(* If simulation of input enabled set it's value to FALSE *)
IF bResetForceValue THEN
	bResetForceValue := FALSE;
	piTestSensor.MR_ResetForceValue();
END_IF

bErrorTimedout := piTestSensor.ErrorTimedout;

bActive 		:= piTestSensor.Active;
CurrentTimeout	:= piTestSensor.CurrentTimeout;

IF bReset THEN
	bReset := FALSE;
	iState := 30;		
END_IF

CASE iState OF 
	0:
		IF bInit THEN
			bInit := FALSE;
			iState := 10;
			
		ELSIF bAbort THEN
			bAbort := FALSE;
			iState := 20;
			
		ELSIF bStartTracking THEN
			bStartTracking := FALSE;
			iState := 40;
			
		END_IF
	10:
		piTestSensor.MR_Init();
		IF piTestSensor.Active THEN
			iState := 0;
		END_IF
		
	20:
		piTestSensor.MR_Abort();
		IF NOT piTestSensor.Active THEN
			iState := 0;
		END_IF
		
	30:
		piTestSensor.MR_Reset();		
		IF NOT piTestSensor.ErrorTimedout THEN
			iState := 0;
		END_IF

	40:
		piTestSensor.MR_StartTracking();
		IF piTestSensor.In OR piTestSensor.ErrorTimedout THEN
			iState := 0;
		END_IF
	
END_CASE

piTestSensor();

END_PROGRAM

// ---- POUs/Universal Blocks/Digital Devices/Digital Output/PRG_FB_DigitalOutput_Test.TcPOU
PROGRAM PRG_FB_DigitalOutput_Test
VAR
	bFirstCycle		: BOOL := TRUE;
	bValue			: BOOL;					(* Output value to set on object *)
	poTestOutput	: FB_DigitalOutput();	(* Digital output object *)
END_VAR

IF bFirstCycle THEN
	bFirstCycle := FALSE;
	poTestOutput.MR_FirstCycle('My test digital output');
END_IF

poTestOutput.Out := bValue;
poTestOutput();

END_PROGRAM

// ---- POUs/Universal Blocks/Digital Devices/Lamp/PRG_FB_Lamp_Test.TcPOU
PROGRAM PRG_FB_Lamp_Test
VAR
	bFirstCycle 	: BOOL := TRUE;
	bTurnOn			: BOOL;				(* Command turn on *)
	bTurnOff		: BOOL;				(* Command turn off *)
	bStartFlashing	: BOOL;				(* Command start flashing *)
	tBlinkTime		: TIME := T#500MS;	(* Blink time *)
	fbLamp 			: FB_Lamp;			(* Lamp object *)
END_VAR

IF bFirstCycle THEN
	bFirstCycle := FALSE;
	fbLamp.MR_FirstCycle('My test lamp');
END_IF

IF bTurnOn THEN
	IF fbLamp.MR_LampOn() THEN
		bTurnOn := FALSE;
	END_IF
	
ELSIF bTurnOff THEN
	IF fbLamp.MR_LampOff() THEN
		bTurnOff := FALSE;
	END_IF
	
ELSIF bStartFlashing THEN
	IF fbLamp.MR_LampBlink(tBlinkTime) THEN
		bStartFlashing := FALSE;
	END_IF
	
END_IF

fbLamp();

END_PROGRAM

// ---- POUs/Universal Blocks/Fixtures/FB_Fixture222.TcPOU
FUNCTION_BLOCK FB_Fixture222 EXTENDS FB_UniversalFixture
VAR_INPUT
END_VAR
VAR_OUTPUT
END_VAR
VAR
	(*
		Add fixture sensors and actuators
	*)
END_VAR

SUPER^();

(*
	Add FB instances
*)

METHOD PROTECTED MS_Close
VAR_INPUT
END_VAR
eFixtureState := UNIVERSAL_FIXTURE_CLOSE_DONE;
END_METHOD

METHOD PROTECTED MS_Open
VAR_INPUT
END_VAR
eFixtureState := UNIVERSAL_FIXTURE_OPEN_DONE;
END_METHOD

METHOD PROTECTED MS_ReadyInitialized
VAR_INPUT
END_VAR
eFixtureState := UNIVERSAL_FIXTURE_IDLE;
END_METHOD

METHOD PROTECTED MS_Reset
VAR_INPUT
END_VAR
eFixtureState := UNIVERSAL_FIXTURE_RESET_DONE;
END_METHOD

PROPERTY SocketOpen : REFERENCE TO BOOL
GET
SocketOpen REF= bSocketOpen;
END_GET
END_PROPERTY

END_FUNCTION_BLOCK

// ---- POUs/Universal Blocks/Fixtures/PRG_FB_FixtureCommTest.TcPOU
PROGRAM PRG_FB_FixtureCommTest
VAR
	bFirstCycle			: BOOL := TRUE;
	
	(* Commands *)
	bInit				: BOOL;
	bMeasure 			: BOOL;
	bAbort				: BOOL;
	bReset				: BOOL;
	bOpen				: BOOL;
	bClose				: BOOL;
	
	(* Parameters *)
	iSampleID			: UINT;
	iState				: INT;
	
	(* Status *)
	bActive				: REFERENCE TO BOOL;
	bSocketOpen			: REFERENCE TO BOOL;
	iCurrentSampleID	: REFERENCE TO UDINT;
	bError				: REFERENCE TO BOOL;
	eFixtureState		: REFERENCE TO E_UniversalFixtureState;
	eResult				: REFERENCE TO E_UniversalFixtureSampleResult;
	
	(* FB's*)
	fbFixtureCommTest	: FB_Fixture;
END_VAR

IF bFirstCycle THEN
	bFirstCycle := FALSE;
	fbFixtureCommTest.MR_FirstCycle( 	sFixtureName 		:= 'PShEll Test Fixture',
										sHost 				:= '192.168.1.1',
										sAmsNetID 			:= '',
										iPort 				:= 12000,
										tTimeout 			:= DEFAULT_ADS_TIMEOUT,
										bUseLogger			:= TRUE,
										bClientConnection 	:= TRUE,
										sLoggerName 		:= 'PShEll Test Fixture',
										sFileDir 			:= 'C:\TwinCAT\Tests\',
										sFileName 			:= 'FixtureCommTest',
										bCreateFileAtStart 	:= TRUE,
										bAddHeader			:= TRUE,
										bAddTimeStamp 		:= TRUE);
	
	(* Update auxilary status variables *)									
	bActive 			REF= fbFixtureCommTest.Active;
	eResult				REF= fbFixtureCommTest.SampleResult;
	bError 				REF= fbFixtureCommTest.Error;
	eFixtureState		REF= fbFixtureCommTest.State;
	iCurrentSampleID	REF= fbFixtureCommTest.SampleID;
	bSocketOpen			REF= fbFixtureCommTest.SocketOpen;
END_IF

IF bReset THEN
	bReset := FALSE;
	iState := 50;
	
ELSIF bAbort THEN
	bAbort := FALSE;
	iState := 60;
	
END_IF

CASE iState OF
	0:
		IF bInit THEN
			bInit := FALSE;
			iState := 10;
			
		ELSIF bMeasure THEN
			bMeasure := FALSE;
			iState := 20;
			
		ELSIF bOpen THEN
			bOpen := FALSE;
			iState := 30;
		
		ELSIF bClose THEN
			bClose := FALSE;
			iState := 40;
			
		END_IF
	10:
		fbFixtureCommTest.MR_Init();
		
		IF fbFixtureCommTest.Active THEN
			iState := 0;
		END_IF
	20:
		fbFixtureCommTest.MR_Measure(iSampleID);
		
		IF NOT fbFixtureCommTest.Busy THEN
			iSampleID := 0;
			iState := 0;
		END_IF
		
	30:
		fbFixtureCommTest.MR_Open();
		
		IF fbFixtureCommTest.SocketOpen THEN
			iState := 0;
		END_IF
		
	40:
		fbFixtureCommTest.MR_Close();
		
		IF NOT fbFixtureCommTest.SocketOpen THEN
			iState := 0;
		END_IF
		
	50:
		fbFixtureCommTest.MR_Reset();
		
		IF NOT fbFixtureCommTest.Error THEN
			iState := 0;
		END_IF
	
	60:
		fbFixtureCommTest.MR_Abort();
		
		IF NOT fbFixtureCommTest.Active THEN
			iState := 0;
		END_IF
	
END_CASE

fbMachineTime(bEnable := TRUE);
fbFixtureCommTest();

END_PROGRAM

// ---- POUs/Universal Blocks/Fixture/FB_Fixture.TcPOU
(*
Copyrights	: Precision Systems Engineering
Author		: ADBO
Date		: 07/2022
Description	: This function block extends standard functionality of FB_FixtureCore with platform pusher and product holder.
*)
FUNCTION_BLOCK FB_Fixture EXTENDS FB_FixtureJig
VAR CONSTANT
	(* Fixture platform cylinder default setup *)
	sCOVER_PUSHER_NAME						: STRING	:= 'Cover Pusher';	(* Platform pusher name *)
	tCOVER_PUSHER_OPEN_TIMEOUT				: TIME 		:= T#5S;			(* Platform pusher opening timeout *)
	tCOVER_PUSHER_CLOSE_TIMEOUT				: TIME 		:= T#5S;			(* Platform pusher closing timeout *)
	tCOVER_PUSHER_MOVE_DELAY 				: TIME 		:= T#0MS;			(* Platform pusher delay after position change *)
	
	(* Fixture product holder default setup *)
	sCLAMP_NAME								: STRING 	:= 'Clamp Pusher';	(* Product holder name *)
	tCLAMP_OPEN_TIMEOUT						: TIME 		:= T#5S;			(* Product holder opening timeout *)
	tCLAMP_CLOSE_TIMEOUT					: TIME 		:= T#5S;			(* Product holder closing timeout *)
	tCLAMP_MOVE_DELAY 						: TIME 		:= T#300MS;//750MS	(* Product holder delay after position change *)
	
	(* Norm loading keywords *)
	sNORM_LOAD_COMMAND						: STRING := 'LDNORM:';			(* Load norm command send from PLC to UTU*)
	sNORM_GSAMPLE_MEASURE_COMMAND			: STRING := 'MeasGSample';		(* Measure Golden sample command send from PLC to UTU after loading new norm *)	
	sNORM_LOAD_SUCCESS 						: STRING := 'OK';				(* Response from UTU: norm loaded successfull *)
	sNORM_LOAD_FAIL							: STRING := 'Fail';				(* Response from UTU: norm load failed *)
	sNORM_GS_REQUEST						: STRING := 'GS:';				(* UTU requests golden sample *)
 	
	(* UTU STATUS *)
	sUTU_STATUS_OK							: STRING := 'OK';
	sUTU_STATUS_NOK							: STRING := 'NOK';
	sUTU_STATUS_bBusy						: STRING := 'bBusy';
	sUTU_STATUS_BCHECKSETUP					: STRING := 'bCheckSetup';
	
	(* Measurement keywords *)
	sMEASUREMENT_START_COMMAND				: STRING := 'bStart$R$N';		(* Start measurement command send from PLC to UTU*)
	
	sMEASUREMENT_BUSY						: STRING := 'bBusy';			(* Response from UTU: measurement started *)
	sMEASUREMENT_FINISHED					: STRING := (*'bReady'; //*)'bDone';			(* Response from UTU: measurement passed *)
	sMEASUREMENT_GOOD_PRODUCT				: STRING := 'bGood';			(* Response from UTU: good product *)
	sMEASUREMENT_REWORK						: STRING := 'bRework';			(* Perform remeasurement of same product *)
	sMEASUREMENT_REMEASURE					: STRING := 'bRemeasure';		(* Perform remeasurement of same product *)
	sMEASUREMENT_ERROR_THD					: STRING := 'bTHDReject';		(* Response from UTU: measurement failed with THD error*)
	sMEASUREMENT_ERROR_PHASE				: STRING := 'bPhaseReject';		(* Response from UTU: measurement failed with PHASE error*)
	sMEASUREMENT_ERROR_SSPL					: STRING := 'bSSPLReject';		(* Response from UTU: measurement failed with SSPL error*)
	sMEASUREMENT_ERROR_RUBBING				: STRING := 'bRubReject';		(* Response from UTU: measurement failed with RUBBING error*)
	sMEASUREMENT_ERROR_IMP					: STRING := 'bImpReject';		(* Response from UTU: measurement failed with INP error*)
	sMEASUREMENT_ERROR_HFA					: STRING := 'bHFAReject';		(* Response from UTU: measurement failed with HFA error*)
	sMEASUREMENT_ERROR_SPL					: STRING := 'bSPLReject';		(* Response from UTU: measurement failed with SPL error*)
	sMEASUREMENT_ERROR_CONNECTION			: STRING := 'bRejectConnect';	(* Response from UTU: measurement failed with connection problems *)
	sMEASUREMENT_ERROR_OTHER				: STRING := 'bReject';			(* Response from UTU: measurement failed *)
	sMEASUREMENT_FINISH_BATCH				: STRING := 'bFinishBatch';		(* Response from UTU: Batch END *)
	sMEASUREMENT_READY						: STRING := 'bReady';
END_VAR
VAR
	(* Auxilary command bits *)
	bCoverActive 							: BOOL;
	bCoverHome 								: BOOL;
	bClampHold 								: BOOL;
	bClampRelease 							: BOOL;
	bCoverActiveAndJigOpen					: BOOL;
	bCoverHomeAndJigClose					: BOOL;
	bLoadNorm								: BOOL;
//	bGSampleMeasure							: BOOL;
//	bGoldenSampelReadyToMeasure				: BOOL;		(* Robot gived Golden sample to Fixture *)
	
	(* Parameters *)
	sProductType							: STRING;
	sProductQuantity						: STRING;
	
	//new
	sConfig									: STRING;
	iAmount									: UINT;
	sPO										: STRING;
	sBatch									: STRING;
	sOPID									: STRING;
	
	(* Status flags *)
	bNormLoaded								: BOOL;
	bBatchEnd								: BOOL;
	bGSampleMeasureRequested				: BOOL;
	bReMeasure								: BOOL;
	bGSampleMeasurmentDone					: BOOL;
	eNormLoadResult							: E_FixtureLoadNormResult;
	eMeasurementResultExt					: E_FixtureMeasurementResultExt;
	
	(* State machines *)
	eFcqFixtureStateInit					: E_FixtureStateInit;
	eFcqFixtureStateAbort					: E_FixtureStateAbort;
	eFcqFixtrueStateReset					: E_FixtureStateReset;
	eFcqFixtureState						: E_FixtureState;
	eFcqFixtureStateLoadNorm				: E_FixtureStateLoadNorm;
	eFcqFixtureStateGSampleMeas				: E_FcqFixtureStateGSampleMeas;
	eFcqFixtureStateMeasurement 			: E_FixtureStateMeasurement;
	eFcqFixtureStateMeasurementDataExchange	: E_FixtureStateMeasurementDataExchange;
	
	eGoldenSampleResult 					: E_GoldenSampleState;
	
	iGsampleId : USINT;
	
	
	(* FB's *)
	fbCover									: FB_DoubleCoilCylinder;		(*  *)
	fbClamp									: FB_FixtureClamp;				(*  *)
	
END_VAR

IF bFirstCycle THEN
	fbCover.MR_FirstCycle(	sName 					:= CONCAT(STR1 :=THIS^.sName, STR2:= sCOVER_PUSHER_NAME),
							sHomeSensorModuleType	:= '?',
							sHomeSensorPortID		:= '?',
							sActiveSensorModuleType	:= '?',
							sActiveSensorPortID		:= '?',
							tGoHomeTimeout 			:= tCOVER_PUSHER_OPEN_TIMEOUT,
							tGoActiveTimeout 		:= tCOVER_PUSHER_CLOSE_TIMEOUT,
							tDelay					:= tCOVER_PUSHER_MOVE_DELAY);
									
	fbClamp.MR_FirstCycle(	sName 					:= CONCAT(STR1 := THIS^.sName, STR2:= sCLAMP_NAME),
							sHomeSensorModuleType	:= '?',
							sHomeSensorPortID		:= '?',
							sActiveSensorModuleType := '?',
							sActiveSensorPortID		:= '?',
							tGoHomeTimeout 			:= tCLAMP_OPEN_TIMEOUT,
							tGoActiveTimeout 		:= tCLAMP_CLOSE_TIMEOUT,
							tDelay					:= tCLAMP_MOVE_DELAY);							
END_IF

(* Run parent main implementation *)
SUPER^();

(* Update status flags*)
bError := bError OR fbClamp.Error OR fbCover.Error;
//IF bError THEN
//	bBusy := FALSE;
//END_IF

(* Run product holder cylinder instance *)
fbClamp();

(* Run fixture platform cylinder instance *)
fbCover();

PROPERTY BatchEnd : REFERENCE TO BOOL
GET
BatchEnd REF= bBatchEnd;
END_GET
END_PROPERTY

PROPERTY ClampHold : REFERENCE TO BOOL
GET
ClampHold REF= fbClamp.PositionActive;
//ClampHold := NOT fbClamp.PositionActive;
END_GET
END_PROPERTY

PROPERTY ClampSimulation : BOOL
GET
ClampSimulation := fbClamp.Simulation;
END_GET
SET
fbClamp.Simulation := ClampSimulation;
END_SET
END_PROPERTY

PROPERTY CoverPositionActive : REFERENCE TO BOOL
GET
CoverPositionActive REF= fbCover.PositionActive;
END_GET
END_PROPERTY

PROPERTY CoverPositionHome : REFERENCE TO BOOL
GET
CoverPositionHome REF= fbCover.PositionHome;
END_GET
END_PROPERTY

PROPERTY CoverSimulation : BOOL
GET
CoverSimulation := fbCover.Simulation;
END_GET
SET
fbCover.Simulation := CoverSimulation;
END_SET
END_PROPERTY

PROPERTY GoldenSampleMeasDone : REFERENCE TO BOOL
GET
GoldenSampleMeasDone REF= bGSampleMeasurmentDone;
END_GET
END_PROPERTY

PROPERTY GoldenSampleMeasRequested : REFERENCE TO BOOL
GET
GoldenSampleMeasRequested REF= bGSampleMeasureRequested;
END_GET
END_PROPERTY

PROPERTY GoldenSampleResult : REFERENCE TO E_GoldenSampleState
GET
GoldenSampleResult REF= eGoldenSampleResult;
END_GET
END_PROPERTY

PROPERTY GSampleId : REFERENCE TO USINT
GET
GSampleId REF= iGsampleId;
END_GET
END_PROPERTY

METHOD PROTECTED M_MeasurementClient : BOOL
VAR_INST
	tonMeasSimulation : TON;
END_VAR
CASE eFixtureStateMeasure OF
	UNIVERSAL_FIXTURE_MEASURE_SEND_DATA:
		sSendData := sMEASUREMENT_START_COMMAND;
		FUN_StringToTcpBufferData(sMessageAddr := ADR(sSendData), stSendDataAddr := ADR(stSendData));
		fbTcpClient.MR_AppendToSendBuffer(stData := stSendData);
		
		eFixtureStateMeasure := UNIVERSAL_FIXTURE_MEASURE_RECIVE_DATA;
		eFcqFixtureStateMeasurementDataExchange := FIXTURE_MEASURE_DATA_EXCHANGING_WAIT_FOR_BUSY;
		
	UNIVERSAL_FIXTURE_MEASURE_RECIVE_DATA:
		stReciveData := fbTcpClient.NextRecivedMessage;
		
		IF stReciveData.iLength > 0 THEN
			FUN_TcpBufferDataToString(sMessageAddr := ADR(sRecivedData), stReturnDataAddr := ADR(stReciveData));
		END_IF
		
			CASE eFcqFixtureStateMeasurementDataExchange OF
				FIXTURE_MEASURE_DATA_EXCHANGING_WAIT_FOR_BUSY:
					IF MEMCMP(ADR(sRecivedData),ADR(sMEASUREMENT_BUSY),INT_TO_UDINT(LEN(sMEASUREMENT_BUSY))) = 0 THEN
						fbTcpClient.MR_ClearReciveBuffer();
						eFcqFixtureStateMeasurementDataExchange := FIXTURE_MEASURE_DATA_EXCHANGING_WAIT_FOR_FISNISH;
					//	eFcqFixtureStateMeasurementDataExchange := FIXTURE_MEASURE_DATA_EXCHANGING_PROCCESS_RESULTS;
					END_IF
				
				FIXTURE_MEASURE_DATA_EXCHANGING_WAIT_FOR_FISNISH:
					IF (MEMCMP(ADR(sRecivedData),ADR(sMEASUREMENT_FINISHED),INT_TO_UDINT(LEN(sMEASUREMENT_FINISHED))) = 0) OR (FIND(sRecivedData,sMEASUREMENT_FINISHED) > 0) THEN
						IF bReMeasure THEN
							fbTcpClient.MR_ClearReciveBuffer();
							eFixtureStateMeasure := UNIVERSAL_FIXTURE_MEASURE_SEND_DATA;
							eFcqFixtureStateMeasurementDataExchange := FIXTURE_MEASURE_DATA_EXCHANGING_WAIT_FOR_BUSY;
						ELSE
							eFcqFixtureStateMeasurementDataExchange := FIXTURE_MEASURE_DATA_EXCHANGING_PROCCESS_RESULTS;
//							eFcqFixtureStateMeasurementDataExchange := FIXTURE_MEASURE_DATA_EXCHANGING_DONE;//
						END_IF	
					END_IF
				
				FIXTURE_MEASURE_DATA_EXCHANGING_PROCCESS_RESULTS:
					(* Good product *)
					IF (MEMCMP(ADR(sRecivedData),ADR(sMEASUREMENT_GOOD_PRODUCT),INT_TO_UDINT(LEN(sMEASUREMENT_GOOD_PRODUCT))) = 0) OR (FIND(sRecivedData,sMEASUREMENT_GOOD_PRODUCT) > 0) THEN
						IF bUseLogger THEN
							sLoggerMessage := CONCAT(sLoggerMessage,sMEASUREMENT_GOOD_PRODUCT);
							fbMeasurementLogger.MR_AddLogs(sLoggerMessage);
						END_IF
						fbTcpClient.MR_ClearReciveBuffer();
						eSampleResult := UNIVERSAL_FIXTURE_SAMPLE_ACCEPTED;
						eMeasurementResultExt := FIXTURE_MEASUREMENT_RESULT_GOOD;
						eFcqFixtureStateMeasurementDataExchange := FIXTURE_MEASURE_DATA_EXCHANGING_DONE;
//						eFcqFixtureStateMeasurementDataExchange := FIXTURE_MEASURE_DATA_EXCHANGING_WAIT_FOR_FISNISH; //

					(* Bad product - rework *)
					ELSIF (MEMCMP(ADR(sRecivedData),ADR(sMEASUREMENT_REWORK),INT_TO_UDINT(LEN(sMEASUREMENT_REWORK))) = 0) OR (FIND(sRecivedData,sMEASUREMENT_REWORK) > 0) THEN
						IF bUseLogger THEN
							sLoggerMessage := CONCAT(sLoggerMessage,sMEASUREMENT_REWORK);
							fbMeasurementLogger.MR_AddLogs(sLoggerMessage);
						END_IF
						fbTcpClient.MR_ClearReciveBuffer();
						eSampleResult := UNIVERSAL_FIXTURE_SAMPLE_REJECTED;
						eMeasurementResultExt := FIXTURE_MEASUREMENT_RESULT_REWORK;
						eFcqFixtureStateMeasurementDataExchange := FIXTURE_MEASURE_DATA_EXCHANGING_DONE;
//						eFcqFixtureStateMeasurementDataExchange := FIXTURE_MEASURE_DATA_EXCHANGING_WAIT_FOR_FISNISH; //
						
						
					(* Bad product - remeaseure *)
					ELSIF (MEMCMP(ADR(sRecivedData),ADR(sMEASUREMENT_REMEASURE),INT_TO_UDINT(LEN(sMEASUREMENT_REMEASURE))) = 0) OR (FIND(sRecivedData,sMEASUREMENT_REMEASURE) > 0) THEN
						fbTcpClient.MR_ClearSendBuffer();
						fbTcpClient.MR_ClearReciveBuffer();
//						bReMeasure := TRUE;
//						eFcqFixtureStateMeasurementDataExchange :=FIXTURE_MEASURE_DATA_EXCHANGING_WAIT_FOR_FISNISH;
						eFixtureStateMeasure := UNIVERSAL_FIXTURE_MEASURE_SEND_DATA;
						eFcqFixtureStateMeasurementDataExchange := FIXTURE_MEASURE_DATA_EXCHANGING_WAIT_FOR_BUSY;
						
					(* Bad product - connection *)	
					ELSIF (MEMCMP(ADR(sRecivedData),ADR(sMEASUREMENT_ERROR_CONNECTION),INT_TO_UDINT(LEN(sMEASUREMENT_ERROR_CONNECTION))) = 0) OR  (FIND(sRecivedData,sMEASUREMENT_ERROR_CONNECTION) > 0)  THEN
						IF bUseLogger THEN
							sLoggerMessage := CONCAT(sLoggerMessage,sMEASUREMENT_ERROR_CONNECTION);
							fbMeasurementLogger.MR_AddLogs(sLoggerMessage);
						END_IF
						fbTcpClient.MR_ClearReciveBuffer();
						eSampleResult := UNIVERSAL_FIXTURE_SAMPLE_REJECTED;
						eMeasurementResultExt := FIXTURE_MEASUREMENT_RESULT_CONNECT;
						eFcqFixtureStateMeasurementDataExchange := FIXTURE_MEASURE_DATA_EXCHANGING_DONE;
//						eFcqFixtureStateMeasurementDataExchange := FIXTURE_MEASURE_DATA_EXCHANGING_WAIT_FOR_FISNISH; //
					
					(* Bad product - THD *)
					ELSIF (MEMCMP(ADR(sRecivedData),ADR(sMEASUREMENT_ERROR_THD),INT_TO_UDINT(LEN(sMEASUREMENT_ERROR_THD))) = 0) OR (FIND(sRecivedData,sMEASUREMENT_ERROR_THD) > 0)  THEN
						IF bUseLogger THEN
							sLoggerMessage := CONCAT(sLoggerMessage,sMEASUREMENT_ERROR_THD);
							fbMeasurementLogger.MR_AddLogs(sLoggerMessage);
						END_IF
						fbTcpClient.MR_ClearReciveBuffer();
						eSampleResult := UNIVERSAL_FIXTURE_SAMPLE_REJECTED;
						eMeasurementResultExt := (*FIXTURE_MEASUREMENT_RESULT_REWORK;*)FIXTURE_MEASUREMENT_RESULT_THD;
						eFcqFixtureStateMeasurementDataExchange := FIXTURE_MEASURE_DATA_EXCHANGING_DONE;
//						eFcqFixtureStateMeasurementDataExchange := FIXTURE_MEASURE_DATA_EXCHANGING_WAIT_FOR_FISNISH; //
					
					(* Bad product - PHASE *)
					ELSIF (MEMCMP(ADR(sRecivedData),ADR(sMEASUREMENT_ERROR_PHASE),INT_TO_UDINT(LEN(sMEASUREMENT_ERROR_PHASE))) = 0) OR (FIND(sRecivedData,sMEASUREMENT_ERROR_PHASE) > 0) THEN
						IF bUseLogger THEN
							sLoggerMessage := CONCAT(sLoggerMessage,sMEASUREMENT_ERROR_PHASE);
							fbMeasurementLogger.MR_AddLogs(sLoggerMessage);
						END_IF
						fbTcpClient.MR_ClearReciveBuffer();
						eSampleResult := UNIVERSAL_FIXTURE_SAMPLE_REJECTED;
						eMeasurementResultExt := FIXTURE_MEASUREMENT_RESULT_PHASE;
						eFcqFixtureStateMeasurementDataExchange := FIXTURE_MEASURE_DATA_EXCHANGING_DONE;
//						eFcqFixtureStateMeasurementDataExchange := FIXTURE_MEASURE_DATA_EXCHANGING_WAIT_FOR_FISNISH; //
					
					(* Bad product - SSPL *)
					ELSIF (MEMCMP(ADR(sRecivedData),ADR(sMEASUREMENT_ERROR_SSPL),INT_TO_UDINT(LEN(sMEASUREMENT_ERROR_SSPL))) = 0) OR (FIND(sRecivedData,sMEASUREMENT_ERROR_SSPL) > 0) THEN
						IF bUseLogger THEN
							sLoggerMessage := CONCAT(sLoggerMessage,sMEASUREMENT_ERROR_SSPL);
							fbMeasurementLogger.MR_AddLogs(sLoggerMessage);
						END_IF
						fbTcpClient.MR_ClearReciveBuffer();
						eSampleResult := UNIVERSAL_FIXTURE_SAMPLE_REJECTED;
						eMeasurementResultExt := FIXTURE_MEASUREMENT_RESULT_SSPL;
						eFcqFixtureStateMeasurementDataExchange := FIXTURE_MEASURE_DATA_EXCHANGING_DONE;
//						eFcqFixtureStateMeasurementDataExchange := FIXTURE_MEASURE_DATA_EXCHANGING_WAIT_FOR_FISNISH; //
					
					(* Bad product - Rubbing *)
					ELSIF (MEMCMP(ADR(sRecivedData),ADR(sMEASUREMENT_ERROR_RUBBING),INT_TO_UDINT(LEN(sMEASUREMENT_ERROR_RUBBING))) = 0) OR (FIND(sRecivedData,sMEASUREMENT_ERROR_RUBBING) > 0) THEN
						IF bUseLogger THEN
							sLoggerMessage := CONCAT(sLoggerMessage,sMEASUREMENT_ERROR_RUBBING);
							fbMeasurementLogger.MR_AddLogs(sLoggerMessage);
						END_IF
						fbTcpClient.MR_ClearReciveBuffer();
						eSampleResult := UNIVERSAL_FIXTURE_SAMPLE_REJECTED;
						eMeasurementResultExt := FIXTURE_MEASUREMENT_RESULT_RUBBING;
						eFcqFixtureStateMeasurementDataExchange := FIXTURE_MEASURE_DATA_EXCHANGING_DONE;
//						eFcqFixtureStateMeasurementDataExchange := FIXTURE_MEASURE_DATA_EXCHANGING_WAIT_FOR_FISNISH; //
					
					(* Bad product - IMP *)
					ELSIF (MEMCMP(ADR(sRecivedData),ADR(sMEASUREMENT_ERROR_IMP),INT_TO_UDINT(LEN(sMEASUREMENT_ERROR_IMP))) = 0) OR (FIND(sRecivedData,sMEASUREMENT_ERROR_IMP) > 0) THEN
						IF bUseLogger THEN
							sLoggerMessage := CONCAT(sLoggerMessage,sMEASUREMENT_ERROR_IMP);
							fbMeasurementLogger.MR_AddLogs(sLoggerMessage);
						END_IF
						fbTcpClient.MR_ClearReciveBuffer();
						eSampleResult := UNIVERSAL_FIXTURE_SAMPLE_REJECTED;
						eMeasurementResultExt := FIXTURE_MEASUREMENT_RESULT_IMP;
						eFcqFixtureStateMeasurementDataExchange := FIXTURE_MEASURE_DATA_EXCHANGING_DONE;
//						eFcqFixtureStateMeasurementDataExchange := FIXTURE_MEASURE_DATA_EXCHANGING_WAIT_FOR_FISNISH; //
					
					(* Bad product - HFA *)
					ELSIF (MEMCMP(ADR(sRecivedData),ADR(sMEASUREMENT_ERROR_HFA),INT_TO_UDINT(LEN(sMEASUREMENT_ERROR_HFA))) = 0) OR (FIND(sRecivedData,sMEASUREMENT_ERROR_HFA) > 0) THEN
						IF bUseLogger THEN
							sLoggerMessage := CONCAT(sLoggerMessage,sMEASUREMENT_ERROR_HFA);
							fbMeasurementLogger.MR_AddLogs(sLoggerMessage);
						END_IF
						fbTcpClient.MR_ClearReciveBuffer();
						eSampleResult := UNIVERSAL_FIXTURE_SAMPLE_REJECTED;
						eMeasurementResultExt := FIXTURE_MEASUREMENT_RESULT_HFA;
						eFcqFixtureStateMeasurementDataExchange := FIXTURE_MEASURE_DATA_EXCHANGING_DONE;
//						eFcqFixtureStateMeasurementDataExchange := FIXTURE_MEASURE_DATA_EXCHANGING_WAIT_FOR_FISNISH; //
						
					(* Bad product - SPL *)
					ELSIF (MEMCMP(ADR(sRecivedData),ADR(sMEASUREMENT_ERROR_OTHER),INT_TO_UDINT(LEN(sMEASUREMENT_ERROR_OTHER))) = 0) OR (FIND(sRecivedData,sMEASUREMENT_ERROR_OTHER) > 0) THEN
						IF bUseLogger THEN
							sLoggerMessage := CONCAT(sLoggerMessage,sMEASUREMENT_ERROR_SPL);
							fbMeasurementLogger.MR_AddLogs(sLoggerMessage);
						END_IF
						fbTcpClient.MR_ClearReciveBuffer();
						eSampleResult := UNIVERSAL_FIXTURE_SAMPLE_REJECTED;
						eMeasurementResultExt := FIXTURE_MEASUREMENT_RESULT_SPL;
						eFcqFixtureStateMeasurementDataExchange := FIXTURE_MEASURE_DATA_EXCHANGING_DONE;
//						eFcqFixtureStateMeasurementDataExchange := FIXTURE_MEASURE_DATA_EXCHANGING_WAIT_FOR_FISNISH; //
					
					ELSIF (MEMCMP(ADR(sRecivedData),ADR(sMEASUREMENT_ERROR_OTHER),INT_TO_UDINT(LEN(sMEASUREMENT_ERROR_OTHER))) = 0) OR (FIND(sRecivedData,sMEASUREMENT_ERROR_OTHER) > 0)  THEN
						IF bUseLogger THEN
							sLoggerMessage := CONCAT(sLoggerMessage,sMEASUREMENT_ERROR_OTHER);
							fbMeasurementLogger.MR_AddLogs(sLoggerMessage);
						END_IF
						fbTcpClient.MR_ClearReciveBuffer();
						eSampleResult := UNIVERSAL_FIXTURE_SAMPLE_REJECTED;
						eMeasurementResultExt := FIXTURE_MEASUREMENT_RESULT_REJECT_OTHER;
						eFcqFixtureStateMeasurementDataExchange := FIXTURE_MEASURE_DATA_EXCHANGING_DONE;
					
					ELSIF (MEMCMP(ADR(sRecivedData),ADR(sMEASUREMENT_READY),INT_TO_UDINT(LEN(sMEASUREMENT_READY))) = 0) OR (FIND(sRecivedData,sMEASUREMENT_READY) > 0)  THEN 
						eFcqFixtureStateMeasurementDataExchange := FIXTURE_MEASURE_DATA_EXCHANGING_DONE;	
					END_IF
					
				FIXTURE_MEASURE_DATA_EXCHANGING_DONE:
					IF (MEMCMP(ADR(sRecivedData),ADR(sMEASUREMENT_READY),INT_TO_UDINT(LEN(sMEASUREMENT_READY))) = 0) OR (FIND(sRecivedData,sMEASUREMENT_READY) > 0) THEN
						eFixtureStateMeasure := UNIVERSAL_FIXTURE_MEASURE_DONE;
					END_IF
			END_CASE		
	//	END_IF
	
	UNIVERSAL_FIXTURE_MEASURE_DONE:
		IF 	(MEMCMP(ADR(sRecivedData),ADR(sMEASUREMENT_FINISH_BATCH),INT_TO_UDINT(LEN(sMEASUREMENT_FINISH_BATCH))) = 0) OR (FIND(sRecivedData,sMEASUREMENT_FINISH_BATCH) > 0) THEN
			bBatchEnd := TRUE;
		END_IF
		fbTcpClient.MR_ClearAllBuffers();
		eFixtureState := UNIVERSAL_FIXTURE_METHOD_DONE;
		
END_CASE
(*
tonMeasSimulation(IN := TRUE, PT := T#2500MS);
IF tonMeasSimulation.Q THEN
	tonMeasSimulation(IN := FALSE);
	eSampleResult := UNIVERSAL_FIXTURE_SAMPLE_ACCEPTED;
	eMeasurementResultExt := FIXTURE_MEASUREMENT_RESULT_GOOD;
	eFixtureState := UNIVERSAL_FIXTURE_METHOD_DONE;
END_IF
*)
END_METHOD

PROPERTY MeasurementResultExt : REFERENCE TO E_FixtureMeasurementResultExt
GET
MeasurementResultExt REF= eMeasurementResultExt;
END_GET
END_PROPERTY

METHOD MR_ClampHold : BOOL
VAR_INPUT
END_VAR
IF eFixtureState = UNIVERSAL_FIXTURE_IDLE AND NOT fbClamp.PositionActive THEN
	bBusy := TRUE;
	bClampHold := TRUE;
	MR_ClampHold := FALSE;
	eFixtureState := UNIVERSAL_FIXTURE_EXTENSION;
	eFcqFixtureState := FIXTURE_EXTENSION_CLAMP_HOLD;
	fbMachineLogger.MR_AddLogs(CONCAT(sName,' : product hold'));
	
ELSIF eFcqFixtureState = FIXTURE_EXTENSION_CLAMP_HOLD_DONE THEN
	bClampHold := FALSE;
	MR_ClampHold := TRUE;
	fbMachineLogger.MR_AddLogs(CONCAT(sName,' : product hold done'));
	
END_IF
END_METHOD

METHOD MR_ClampRelease : BOOL
VAR_INPUT
END_VAR
IF eFixtureState = UNIVERSAL_FIXTURE_IDLE AND fbClamp.PositionActive THEN
	bBusy := TRUE;
	bClampRelease := TRUE;
	MR_ClampRelease := FALSE;
	eFixtureState := UNIVERSAL_FIXTURE_EXTENSION;
	eFcqFixtureState := FIXTURE_EXTENSION_CLAMP_RELEASE;
	fbMachineLogger.MR_AddLogs(CONCAT(sName,' : product release'));
	
ELSIF eFcqFixtureState = FIXTURE_EXTENSION_CLAMP_RELEASE_DONE THEN
	bClampRelease := FALSE;
	MR_ClampRelease := TRUE;
	fbMachineLogger.MR_AddLogs(CONCAT(sName,' : product release done'));
	
END_IF
END_METHOD

METHOD MR_CoverActive : BOOL
VAR_INPUT
END_VAR
IF eFixtureState = UNIVERSAL_FIXTURE_IDLE AND NOT fbCover.PositionActive THEN
	bBusy := TRUE;
	bCoverActive := TRUE;
	MR_CoverActive := FALSE;
	eFixtureState := UNIVERSAL_FIXTURE_EXTENSION;
	eFcqFixtureState := FIXTURE_EXTENSION_COVER_ACTIVE;
	fbMachineLogger.MR_AddLogs(CONCAT(sName,' : platform go active'));
	
ELSIF eFcqFixtureState = FIXTURE_EXTENSION_COVER_ACTIVE_DONE THEN
	bCoverActive := FALSE;
	MR_CoverActive := TRUE;
	fbMachineLogger.MR_AddLogs(CONCAT(sName,' : platform go active done'));
	
END_IF
END_METHOD

METHOD MR_CoverActiveAndJigOpen : BOOL
VAR_INPUT
END_VAR
//IF eFixtureState = UNIVERSAL_FIXTURE_IDLE AND (NOT fbCover.PositionActive AND NOT THIS^.SocketOpen) THEN
IF eFixtureState = UNIVERSAL_FIXTURE_IDLE AND (NOT fbCover.PositionActive OR NOT THIS^.SocketOpen) THEN
	bBusy := TRUE;
	bCoverActiveAndJigOpen := TRUE;
	MR_CoverActiveAndJigOpen := FALSE;
	eFixtureState := UNIVERSAL_FIXTURE_EXTENSION;
	eFcqFixtureState := FIXTURE_EXTENSION_COVER_ACTIVE_AND_JIG_OPEN;
	fbMachineLogger.MR_AddLogs(CONCAT(sName,' : platform go active and open'));
	
ELSIF eFcqFixtureState = FIXTURE_EXTENSION_COVER_ACTIVE_AND_JIG_OPEN_DONE THEN
	bCoverActiveAndJigOpen := FALSE;
	MR_CoverActiveAndJigOpen := TRUE;
	fbMachineLogger.MR_AddLogs(CONCAT(sName,' : platform go active and open done'));
	
END_IF
END_METHOD

METHOD MR_CoverHome : BOOL
VAR_INPUT
END_VAR
IF eFixtureState = UNIVERSAL_FIXTURE_IDLE AND NOT fbCover.PositionHome THEN
	bBusy := TRUE;
	bCoverHome := TRUE;
	MR_CoverHome := FALSE;
	eFixtureState := UNIVERSAL_FIXTURE_EXTENSION;
	eFcqFixtureState := FIXTURE_EXTENSION_COVER_HOME;
	fbMachineLogger.MR_AddLogs(CONCAT(sName,' : platform go home'));
	
ELSIF eFcqFixtureState = FIXTURE_EXTENSION_COVER_HOME_DONE THEN
	bCoverHome := FALSE;
	MR_CoverHome := TRUE;
	fbMachineLogger.MR_AddLogs(CONCAT(sName,' : platform go home done'));
	
END_IF
END_METHOD

METHOD MR_CoverHomeAndJigClose : BOOL
VAR_INPUT
END_VAR
//IF eFixtureState = UNIVERSAL_FIXTURE_IDLE AND NOT fbCover.PositionHome AND THIS^.SocketOpen THEN
IF eFixtureState = UNIVERSAL_FIXTURE_IDLE AND (NOT fbCover.PositionHome OR THIS^.SocketOpen) THEN
	bBusy := TRUE;
	bCoverHomeAndJigClose := TRUE;
	MR_CoverHomeAndJigClose := FALSE;
	eFixtureState := UNIVERSAL_FIXTURE_EXTENSION;
	eFcqFixtureState := FIXTURE_EXTENSION_COVER_HOME_AND_JIG_CLOSE;
	fbMachineLogger.MR_AddLogs(CONCAT(sName,' : platform go home and close'));
	
ELSIF eFcqFixtureState = FIXTURE_EXTENSION_COVER_HOME_AND_JIG_CLOSE_DONE THEN
	bCoverHomeAndJigClose := FALSE;
	MR_CoverHomeAndJigClose := TRUE;
	fbMachineLogger.MR_AddLogs(CONCAT(sName,' : platform go home and close done'));
	
END_IF
END_METHOD

METHOD MR_GSampleMeas : BOOL
VAR_INPUT
END_VAR
//IF eNormLoadResult = FIXTURE_NORM_LOAD_GOLDEN_SAMPLE_NEEDED AND eFcqFixtureStateLoadNorm = FIXTURE_LOADING_NORM_GOLDEN_SAMPLE_WAIT_FOR_END THEN
IF eNormLoadResult = FIXTURE_NORM_LOAD_GOLDEN_SAMPLE_NEEDED AND eFixtureState = UNIVERSAL_FIXTURE_IDLE THEN
	bBusy := TRUE;
	bGSampleMeasurmentDone := FALSE;	
	MR_GSampleMeas := FALSE;
//	bGSampleMeasure := TRUE;
	eGoldenSampleResult := GS_STATUS_UNKNOWN;
	eFixtureState := UNIVERSAL_FIXTURE_EXTENSION;
	eFcqFixtureState := FIXTURE_EXTENSION_GOLDEN_SAMPLE_MEASURE;
	eFcqFixtureStateGSampleMeas := FIXTURE_GOLDEN_SAMPLE_SEND_MEASURE_COMMAND;
	fbMachineLogger.MR_AddLogs(CONCAT(sName,' : Golden Sample measurment requested'));
	
	
ELSIF eFcqFixtureState = FIXTURE_EXTENSION_GOLDEN_SAMPLE_MEASURE_DONE THEN
	bBusy := FALSE;
	MR_GSampleMeas := TRUE;
	eFixtureState := UNIVERSAL_FIXTURE_EXTENSION;
	eFcqFixtureState := FIXTURE_EXTENSION_LOAD_NORM;
	//eFcqFixtureStateLoadNorm := FIXTURE_LOADING_NORM_WAIT_FOR_RESPONSE;
	//fbMachineLogger.MR_AddLogs(CONCAT(sName,' : Golden Sample  '));
	fbMachineLogger.MR_AddLogs(CONCAT(sName,CONCAT(' : Golden Sample ID: ',CONCAT(UDINT_TO_STRING(iGsampleId),' measurment done'))));
	bGSampleMeasurmentDone := TRUE;
END_IF
END_METHOD

METHOD MR_LoadNorm : BOOL
VAR_INPUT
	sConfig				: STRING;
	iAmount				: UINT;
	sPO					: STRING;
	sBatch				: STRING;
	sOPID				: STRING;
//	sProductType 		: STRING;	(* Name of product possesed from MES*)
//	sProductQuantity	: STRING;	(* Product quantity *)
END_VAR
IF eFixtureState = UNIVERSAL_FIXTURE_IDLE THEN
	THIS^.sConfig := sConfig;
	THIS^.iAmount := iAmount;
	THIS^.sPO := sPO;
	THIS^.sBatch := sBatch;
	THIS^.sOPID := sOPID;
	
(*	OLD
	THIS^.sProductType := sProductType;
	THIS^.sProductQuantity := sProductQuantity;
*)	
	bNormLoaded := FALSE;
	eNormLoadResult := FIXTURE_NORM_LOAD_UNKNOWN;
//	bLoadNorm := TRUE;
	MR_LoadNorm := FALSE;
	eFixtureState := UNIVERSAL_FIXTURE_EXTENSION;
	eFcqFixtureState := FIXTURE_EXTENSION_LOAD_NORM;
	eFcqFixtureStateLoadNorm := FIXTURE_LOADING_NORM_SEND_NORM_DATA;
	fbMachineLogger.MR_AddLogs(CONCAT(sName,' : load norm requested'));
	
ELSIF eFcqFixtureState = FIXTURE_EXTENSION_LOAD_NORM_DONE THEN
	bNormLoaded := (*NOT bGSampleMeasureRequested;//*)TRUE;
	MR_LoadNorm := TRUE;
	fbMachineLogger.MR_AddLogs(CONCAT(sName,' : norm loaded '));
	
END_IF
END_METHOD

METHOD MR_Reset : BOOL
VAR_INPUT
END_VAR
IF eFixtureState = UNIVERSAL_FIXTURE_METHOD_DONE THEN
	eFcqFixtrueStateReset:=FIXTURE_RESET_CLAMP;
END_IF
SUPER^.MR_Reset();
END_METHOD

METHOD PROTECTED MS_Aborting
VAR_INPUT
END_VAR
CASE eFcqFixtureStateAbort OF
	FIXTURE_ABORT_CLAMP:
		fbClamp.MR_Abort();
		IF NOT fbClamp.Active THEN
			eFcqFixtureStateAbort := FIXTURE_ABORT_COVER;
		END_IF
		
	FIXTURE_ABORT_COVER:
		fbCover.MR_Abort();
		IF NOT fbCover.Active THEN
			eJigStateAbort := FIXTURE_JIG_ABORT_JIG_PUSHER;
			eFcqFixtureStateAbort := FIXTURE_ABORT_DONE;
		END_IF
		
	FIXTURE_ABORT_DONE:
		SUPER^.MS_Aborting();
		
END_CASE
END_METHOD

METHOD MS_ClampHold
VAR_INPUT
END_VAR
fbClamp.MR_GoActive();
IF fbClamp.PositionActive AND NOT fbClamp.Busy THEN
	eFcqFixtureState := FIXTURE_EXTENSION_CLAMP_HOLD_DONE;
END_IF
END_METHOD

METHOD MS_ClampHoldDone
VAR_INPUT
END_VAR
IF NOT bClampHold THEN
	bBusy := FALSE;
	eFixtureState := UNIVERSAL_FIXTURE_IDLE;
	eFcqFixtureState := FIXTURE_EXTENSION_IDLE;
END_IF
END_METHOD

METHOD MS_ClampRelease
VAR_INPUT
END_VAR
fbClamp.MR_GoHome();
IF NOT fbClamp.PositionActive AND NOT fbClamp.Busy THEN
	eFcqFixtureState := FIXTURE_EXTENSION_CLAMP_RELEASE_DONE;
END_IF
END_METHOD

METHOD MS_ClampReleaseDone
VAR_INPUT
END_VAR
IF NOT bClampRelease THEN
	bBusy := FALSE;
	eFixtureState := UNIVERSAL_FIXTURE_IDLE;
	eFcqFixtureState := FIXTURE_EXTENSION_IDLE;
END_IF
END_METHOD

METHOD MS_CoverActive
VAR_INPUT
END_VAR
fbCover.MR_GoActive();
IF fbCover.PositionActive AND NOT fbCover.Busy THEN
	eFcqFixtureState := FIXTURE_EXTENSION_COVER_ACTIVE_DONE;
END_IF
END_METHOD

METHOD MS_CoverActiveAndJigOpen : BOOL
VAR_INPUT
END_VAR
fbCover.MR_GoActive();
fbJig.MR_GoActive();
IF fbCover.PositionActive AND NOT fbCover.Busy AND
	fbJig.PositionActive AND NOT fbJig.Busy THEN
	eFcqFixtureState := FIXTURE_EXTENSION_COVER_ACTIVE_AND_JIG_OPEN_DONE;
END_IF
END_METHOD

METHOD MS_CoverActiveAndJigOpenDone : BOOL
VAR_INPUT
END_VAR
IF NOT bCoverActiveAndJigOpen THEN
	bBusy := FALSE;
	eFixtureState := UNIVERSAL_FIXTURE_IDLE;
	eFcqFixtureState := FIXTURE_EXTENSION_IDLE;
END_IF
END_METHOD

METHOD MS_CoverActiveDone
VAR_INPUT
END_VAR
IF NOT bCoverActive THEN
	bBusy := FALSE;
	eFixtureState := UNIVERSAL_FIXTURE_IDLE;
	eFcqFixtureState := FIXTURE_EXTENSION_IDLE;
END_IF
END_METHOD

METHOD MS_CoverHome
VAR_INPUT
END_VAR
fbCover.MR_GoHome();
IF fbCover.PositionHome AND NOT fbCover.Busy THEN
	eFcqFixtureState := FIXTURE_EXTENSION_COVER_HOME_DONE;
END_IF
END_METHOD

METHOD MS_CoverHomeAndJigClose : BOOL
VAR_INPUT
END_VAR
fbCover.MR_GoHome();
fbJig.MR_GoHome();
IF fbCover.PositionHome AND NOT fbCover.Busy AND
	fbJig.PositionHome AND NOT fbJig.Busy THEN
	eFcqFixtureState := FIXTURE_EXTENSION_COVER_HOME_AND_JIG_CLOSE_DONE;
END_IF
END_METHOD

METHOD MS_CoverHomeAndJigCloseDone : BOOL
VAR_INPUT
END_VAR
IF NOT bCoverHomeAndJigClose THEN
	bBusy := FALSE;
	eFixtureState := UNIVERSAL_FIXTURE_IDLE;
	eFcqFixtureState := FIXTURE_EXTENSION_IDLE;
END_IF
END_METHOD

METHOD MS_CoverHomeDone
VAR_INPUT
END_VAR
IF NOT bCoverHome THEN
	bBusy := FALSE;
	eFixtureState := UNIVERSAL_FIXTURE_IDLE;
	eFcqFixtureState := FIXTURE_EXTENSION_IDLE;
END_IF
END_METHOD

METHOD PROTECTED MS_Extension
VAR_INPUT
END_VAR
CASE eFcqFixtureState OF
	E_FixtureState.FIXTURE_EXTENSION_IDLE:
		bBusy := FALSE;
		
	E_FixtureState.FIXTURE_EXTENSION_COVER_ACTIVE:
		MS_CoverActive();
		
	E_FixtureState.FIXTURE_EXTENSION_COVER_ACTIVE_DONE:
		MS_CoverActiveDone();
		
	E_FixtureState.FIXTURE_EXTENSION_COVER_HOME:
		MS_CoverHome();
		
	E_FixtureState.FIXTURE_EXTENSION_COVER_HOME_DONE:
		MS_CoverHomeDone();	
	
	E_FixtureState.FIXTURE_EXTENSION_CLAMP_HOLD:
		MS_ClampHold();
		
	E_FixtureState.FIXTURE_EXTENSION_CLAMP_HOLD_DONE:
		MS_ClampHoldDone();
		
	E_FixtureState.FIXTURE_EXTENSION_CLAMP_RELEASE:
		MS_ClampRelease();
		
	E_FixtureState.FIXTURE_EXTENSION_CLAMP_RELEASE_DONE:
		MS_ClampReleaseDone();
	
	FIXTURE_EXTENSION_COVER_ACTIVE_AND_JIG_OPEN:
		MS_CoverActiveAndJigOpen();
		
	FIXTURE_EXTENSION_COVER_ACTIVE_AND_JIG_OPEN_DONE:
		MS_CoverActiveAndJigOpenDone();
		
	FIXTURE_EXTENSION_COVER_HOME_AND_JIG_CLOSE:
		MS_CoverHomeAndJigClose();
		
	FIXTURE_EXTENSION_COVER_HOME_AND_JIG_CLOSE_DONE:
		MS_CoverHomeAndJigCloseDone();
		
	FIXTURE_EXTENSION_LOAD_NORM:
		MS_LoadNorm();
		
	FIXTURE_EXTENSION_LOAD_NORM_DONE:
		MS_LoadNormDone();
		
	FIXTURE_EXTENSION_GOLDEN_SAMPLE_MEASURE:	
		MS_GSampleMeas();
		
	FIXTURE_EXTENSION_GOLDEN_SAMPLE_MEASURE_DONE:
		MS_GSampleMeasDone();
	
END_CASE
END_METHOD

METHOD MS_GSampleMeas : BOOL
bBusy := MEMCMP(ADR(sRecivedData),ADR(sUTU_STATUS_bBusy),INT_TO_UDINT(LEN(sUTU_STATUS_bBusy))) = 0; (*	UTU busy flags *)	
CASE eFcqFixtureStateGSampleMeas OF
	//FIXTURE_GOLDEN_SAMPLE_CLOSE:
	//	fbJig.MR_GoActive();
	//	IF fbJig.PositionActive AND NOT fbJig.Busy THEN
	//		eFcqFixtureStateGSampleMeas := FIXTURE_GOLDEN_SAMPLE_SEND_MEASURE_COMMAND;
	//	END_IF
	
	FIXTURE_GOLDEN_SAMPLE_SEND_MEASURE_COMMAND:
		sSendData := sNORM_GSAMPLE_MEASURE_COMMAND;
		sSendData := CONCAT(sSendData, '$R$N');
		FUN_StringToTcpBufferData(sMessageAddr := ADR(sSendData), stSendDataAddr := ADR(stSendData));
		fbTcpClient.MR_AppendToSendBuffer(stData := stSendData);
		eFcqFixtureStateGSampleMeas := FIXTURE_GOLDEN_SAMPLE_WAIT_FOR_RESPONSE;
		
	FIXTURE_GOLDEN_SAMPLE_WAIT_FOR_RESPONSE:
		stReciveData := fbTcpClient.NextRecivedMessage;
		IF stReciveData.iLength > 0 THEN
			FUN_TcpBufferDataToString(sMessageAddr := ADR(sRecivedData), stReturnDataAddr := ADR(stReciveData));
			(* UTU returns bCheckSetup *)
			IF (MEMCMP(ADR(sRecivedData),ADR(sUTU_STATUS_BCHECKSETUP),INT_TO_UDINT(LEN(sUTU_STATUS_BCHECKSETUP))) = 0) THEN
				IF bUseLogger THEN
					sLoggerMessage := CONCAT(sLoggerMessage,sUTU_STATUS_BCHECKSETUP);
					fbMeasurementLogger.MR_AddLogs(sLoggerMessage);
				END_IF
				eGoldenSampleResult := GS_STATUS_BCHECKSETUP;
				//eNormLoadResult := FIXTURE_NORM_LOAD_FAIL;
				eFcqFixtureStateGSampleMeas := FIXTURE_GOLDEN_SAMPLE_MEASUREMENT_DONE; 
			(* UTU returns NOK *)	
			ELSIF (MEMCMP(ADR(sRecivedData),ADR(sUTU_STATUS_NOK),INT_TO_UDINT(LEN(sUTU_STATUS_NOK))) = 0) THEN
				eFcqFixtureStateGSampleMeas := FIXTURE_GOLDEN_SAMPLE_WAIT_FOR_UTU;
				eGoldenSampleResult := GS_STATUS_NOK;
			(* UTU returns OK *)		
			ELSIF (MEMCMP(ADR(sRecivedData),ADR(sUTU_STATUS_OK),INT_TO_UDINT(LEN(sUTU_STATUS_OK))) = 0) THEN
				IF bUseLogger THEN
					sLoggerMessage := CONCAT(sLoggerMessage,sSAMPLE_ACCEPTED);
					fbMeasurementLogger.MR_AddLogs(sLoggerMessage);
				END_IF
				eGoldenSampleResult := GS_STATUS_OK;
				eFcqFixtureStateGSampleMeas := FIXTURE_GOLDEN_SAMPLE_MEASUREMENT_DONE;		
			END_IF
		END_IF
		
(*	FIXTURE_GOLDEN_SAMPLE_OPEN:
		fbJig.MR_GoHome();
		IF (fbJig.PositionHome AND NOT fbJig.Busy) AND NOT fbCover.PositionHome THEN
 			fbClamp.MR_GoHome(); 			
		ELSE
			fbClamp.MR_GoActive();
		END_IF
		IF fbJig.PositionHome AND fbClamp.PositionHome THEN
			fbCover.MR_GoHome();
		END_IF
				
		IF fbClamp.PositionActive AND NOT fbClamp.Busy AND fbCover.PositionHome AND NOT fbCover.Busy AND 
			fbJig.PositionHome AND NOT fbJig.Busy THEN
			eFcqFixtureStateGSampleMeas := FIXTURE_GOLDEN_SAMPLE_MEASUREMENT_DONE;
		ELSE eFcqFixtureStateGSampleMeas := FIXTURE_GOLDEN_SAMPLE_OPEN;
		END_IF
*)
	FIXTURE_GOLDEN_SAMPLE_WAIT_FOR_UTU:
		stReciveData := fbTcpClient.NextRecivedMessage;
		IF stReciveData.iLength > 0 THEN
			FUN_TcpBufferDataToString(sMessageAddr := ADR(sRecivedData), stReturnDataAddr := ADR(stReciveData));
			IF (MEMCMP(ADR(sRecivedData),ADR(sUTU_STATUS_BCHECKSETUP),INT_TO_UDINT(LEN(sUTU_STATUS_BCHECKSETUP))) = 0) THEN
				IF bUseLogger THEN
					sLoggerMessage := CONCAT(sLoggerMessage,sUTU_STATUS_BCHECKSETUP);
					fbMeasurementLogger.MR_AddLogs(sLoggerMessage);
				END_IF
				eGoldenSampleResult := GS_STATUS_BCHECKSETUP;
				//eNormLoadResult := FIXTURE_NORM_LOAD_FAIL;
				eFcqFixtureStateGSampleMeas := FIXTURE_GOLDEN_SAMPLE_MEASUREMENT_DONE; 
			(* UTU returns bCheckSetup *)
			ELSIF (MEMCMP(ADR(sRecivedData),ADR(sNORM_GS_REQUEST),INT_TO_UDINT(LEN(sNORM_GS_REQUEST))) = 0) OR (FIND(sRecivedData,sNORM_GS_REQUEST) > 0) THEN
				bGSampleMeasureRequested := TRUE;
				iGsampleId := STRING_TO_USINT(LEFT(RIGHT(sRecivedData,2),1));
				IF bUseLogger THEN
					sLoggerMessage := CONCAT(sLoggerMessage,'Golden Sample Test');
					fbMeasurementLogger.MR_AddLogs(sLoggerMessage);
				END_IF
				eFcqFixtureStateGSampleMeas := FIXTURE_GOLDEN_SAMPLE_MEASUREMENT_DONE;
			END_IF
		END_IF	
		
	FIXTURE_GOLDEN_SAMPLE_MEASUREMENT_DONE:
		eFcqFixtureState := FIXTURE_EXTENSION_GOLDEN_SAMPLE_MEASURE_DONE;
		
END_CASE
END_METHOD

METHOD MS_GSampleMeasDone : BOOL
VAR_INPUT
END_VAR
bBusy := FALSE;
//eFixtureState := UNIVERSAL_FIXTURE_EXTENSION;
//eFcqFixtureState := FIXTURE_EXTENSION_LOAD_NORM;
//eFcqFixtureStateLoadNorm := FIXTURE_LOADING_NORM_WAIT_FOR_RESPONSE;
eFixtureState := UNIVERSAL_FIXTURE_IDLE;
eFcqFixtureState := FIXTURE_EXTENSION_IDLE;
bGSampleMeasurmentDone := TRUE;
END_METHOD

METHOD PROTECTED MS_Initializing
VAR_INPUT
END_VAR
CASE eFcqFixtureStateInit OF
	FIXTURE_INIT_CLAMP:
		fbClamp.MR_Init();
		
		IF fbClamp.Active THEN
			eFcqFixtureStateInit := FIXTURE_INIT_COVER;
		END_IF
		
	FIXTURE_INIT_COVER:
		fbCover.MR_Init();
		
		IF fbCover.Active THEN
			eJigStateInit := FIXTURE_JIG_INIT_JIG_PUSHER;
			eFcqFixtureStateInit := FIXTURE_INIT_DONE;
		END_IF
		
	FIXTURE_INIT_DONE:
		SUPER^.MS_Initializing();
		
END_CASE
END_METHOD

METHOD MS_LoadNorm
VAR_INST
	TestTON :	TON;
END_VAR
bBusy := MEMCMP(ADR(sRecivedData),ADR(sUTU_STATUS_bBusy),INT_TO_UDINT(LEN(sUTU_STATUS_bBusy))) = 0; (*	UTU busy flags *)	

		
CASE eFcqFixtureStateLoadNorm OF
	FIXTURE_LOADING_NORM_SEND_NORM_DATA:
		(* Prepare and send data to client *)
		sSendData := CONCAT(STR1 := sNORM_LOAD_COMMAND, 
			STR2 :=	CONCAT(STR1 := sConfig,STR2 := CONCAT(STR1 := ':', 
			STR2 := CONCAT(STR1 := UINT_TO_STRING(iAmount),	STR2 := CONCAT(STR1 := ':',
			STR2 := CONCAT(STR1:= sPO, STR2:= CONCAT(STR1:= ':', 
			STR2 := CONCAT(STR1 := sBatch, STR2 := CONCAT(STR1:= ':',
			STR2 := CONCAT(STR1:=sOPID, STR2:= ':'))))))))));
		
		sSendData := CONCAT(sSendData, '$R$N');
		FUN_StringToTcpBufferData(sMessageAddr := ADR(sSendData), stSendDataAddr := ADR(stSendData));
		fbTcpClient.MR_AppendToSendBuffer(stData := stSendData);
		
		(* Prepare data for logger *)
		IF bUseLogger THEN
			MEMSET(ADR(sLoggerMessage),0,INT_TO_UDINT(LEN(sLoggerMessage)));
			sLoggerMessage := CONCAT(STR1 := 'Load norm request:',STR2 := CONCAT(STR1 := sProductType,STR2 := (*USINT_TO_STRING*)(sProductQuantity)));
		END_IF
		
		eFcqFixtureStateLoadNorm := FIXTURE_LOADING_NORM_WAIT_FOR_RESPONSE;
		
	FIXTURE_LOADING_NORM_WAIT_FOR_RESPONSE:
		stReciveData := fbTcpClient.NextRecivedMessage;
		IF stReciveData.iLength > 0  THEN
		FUN_TcpBufferDataToString(sMessageAddr := ADR(sRecivedData), stReturnDataAddr := ADR(stReciveData));
		(* Norm loading Gold Sample *)
			IF (MEMCMP(ADR(sRecivedData),ADR(sNORM_GS_REQUEST),INT_TO_UDINT(LEN(sNORM_GS_REQUEST))) = 0) OR (FIND(sRecivedData,sNORM_GS_REQUEST) > 0) THEN
				iSampleID := STRING_TO_USINT(LEFT(RIGHT(sRecivedData,2),1));
				bGSampleMeasureRequested := TRUE;
				IF bUseLogger THEN
					sLoggerMessage := CONCAT(sLoggerMessage,'Golden Sample Test');
					fbMeasurementLogger.MR_AddLogs(sLoggerMessage);
				END_IF
				
				bGSampleMeasurmentDone := FALSE;
				bBusy := FALSE;
				eNormLoadResult := FIXTURE_NORM_LOAD_GOLDEN_SAMPLE_NEEDED;
				eFcqFixtureStateLoadNorm := FIXTURE_LOADING_NORM_DONE;
				
//			eFcqFixtureStateLoadNorm :=FIXTURE_LOADING_NORM_GOLDEN_SAMPLE_TEST;
							
//			ELSIF MEMCMP(ADR(sRecivedData),ADR(sUTU_STATUS_NOK),INT_TO_UDINT(LEN(sUTU_STATUS_NOK))) = 0 THEN
//				IF bUseLogger THEN
//					sLoggerMessage := CONCAT(sLoggerMessage,CONCAT('golden sample ID:',CONCAT(USINT_TO_STRING(iGsampleId),'	NOK')));
//					fbMeasurementLogger.MR_AddLogs(sLoggerMessage);
//				END_IF
				
			(* Norm loading successfull *)
			ELSIF MEMCMP(ADR(sRecivedData),ADR(sNORM_LOAD_SUCCESS),INT_TO_UDINT(LEN(sNORM_LOAD_SUCCESS))) = 0 THEN
				IF bUseLogger THEN
					sLoggerMessage := CONCAT(sLoggerMessage,sSAMPLE_ACCEPTED);
					fbMeasurementLogger.MR_AddLogs(sLoggerMessage);
				END_IF
				bGSampleMeasureRequested := FALSE;
				bBusy := FALSE;
				eNormLoadResult := FIXTURE_NORM_LOAD_SUCCESS;
				eFcqFixtureStateLoadNorm := FIXTURE_LOADING_NORM_DONE;
				
				
			(* Norm loading failed *)
			ELSIF (MEMCMP(ADR(sRecivedData),ADR(sNORM_LOAD_FAIL),INT_TO_UDINT(LEN(sNORM_LOAD_FAIL))) = 0) THEN
				IF bUseLogger THEN
					sLoggerMessage := CONCAT(sLoggerMessage,sSAMPLE_REJECTED);
					fbMeasurementLogger.MR_AddLogs(sLoggerMessage);
				END_IF
				bGSampleMeasureRequested := FALSE;
				bBusy := FALSE;
				eNormLoadResult := FIXTURE_NORM_LOAD_FAIL;
				eFcqFixtureStateLoadNorm := FIXTURE_LOADING_NORM_DONE;
			
			(* UTU returns bCheckSetup *)
			ELSIF (MEMCMP(ADR(sRecivedData),ADR(sUTU_STATUS_BCHECKSETUP),INT_TO_UDINT(LEN(sUTU_STATUS_BCHECKSETUP))) = 0) THEN
				IF bUseLogger THEN
					sLoggerMessage := CONCAT(sLoggerMessage,sUTU_STATUS_BCHECKSETUP);
					fbMeasurementLogger.MR_AddLogs(sLoggerMessage);
				END_IF
				bGSampleMeasureRequested := FALSE;
				bBusy := FALSE;
				eNormLoadResult := FIXTURE_NORM_LOAD_FAIL;
				eFcqFixtureStateLoadNorm := FIXTURE_LOADING_NORM_DONE;
			END_IF
		END_IF
			
	FIXTURE_LOADING_NORM_DONE:
		fbTcpClient.MR_ClearAllBuffers();
		eFcqFixtureState := FIXTURE_EXTENSION_LOAD_NORM_DONE;
		
END_CASE
END_METHOD

METHOD MS_LoadNormDone
VAR_INPUT
END_VAR
IF NOT bLoadNorm THEN
	bBusy := FALSE;
	bBatchEnd := FALSE;
	eFixtureState := UNIVERSAL_FIXTURE_IDLE;
	eFcqFixtureState := FIXTURE_EXTENSION_IDLE;
END_IF
END_METHOD

METHOD PROTECTED MS_MethodDone
VAR_INPUT
END_VAR
bBusy := FALSE;
SUPER^.MS_MethodDone();
END_METHOD

METHOD PROTECTED MS_Ready
VAR_INPUT
END_VAR
eFcqFixtureStateInit := FIXTURE_INIT_CLAMP;
eFixtureState := UNIVERSAL_FIXTURE_IDLE;
END_METHOD

METHOD PROTECTED MS_Reset
VAR_INPUT
END_VAR
CASE eFcqFixtrueStateReset OF
	FIXTURE_RESET_CLAMP:
		fbClamp.MR_Reset();
		
		IF NOT fbClamp.Error THEN
			eFcqFixtrueStateReset := FIXTURE_RESET_COVER;
		END_IF
		
	FIXTURE_RESET_COVER:
		fbCover.MR_Reset();
		
		IF NOT fbCover.Error THEN
			eJigStateReset := FIXTURE_JIG_RESET_JIG_PUSHER;
			eFcqFixtrueStateReset := FIXTURE_RESET_DONE;
		END_IF
	
	FIXTURE_RESET_DONE:
		SUPER^.MS_Reset();
	
END_CASE
END_METHOD

METHOD PROTECTED MS_Uninitialized
VAR_INPUT
END_VAR
bNormLoaded := FALSE;

SUPER^.MS_Uninitialized();
END_METHOD

PROPERTY NormLoaded : REFERENCE TO BOOL
GET
NormLoaded REF= bNormLoaded;
END_GET
END_PROPERTY

PROPERTY NormLoadResults : REFERENCE TO E_FixtureLoadNormResult
GET
NormLoadResults REF= eNormLoadResult;
END_GET
END_PROPERTY

PROPERTY ref_Clamp : REFERENCE TO FB_FixtureClamp
GET
ref_Clamp REF= fbClamp;
END_GET
END_PROPERTY

PROPERTY ref_Cover : REFERENCE TO FB_DoubleCoilCylinder
GET
ref_Cover REF= fbCover;
END_GET
END_PROPERTY

PROPERTY StateExt : REFERENCE TO E_FixtureState
GET
StateExt REF= eFcqFixtureState;
END_GET
END_PROPERTY

METHOD PROTECTED StateMachine
VAR_INPUT
END_VAR
SUPER^.StateMachine();

CASE eFcqFixtureState OF
	E_FixtureState.FIXTURE_EXTENSION_COVER_ACTIVE:
		MS_CoverActive();
		
	E_FixtureState.FIXTURE_EXTENSION_COVER_ACTIVE_DONE:
		MS_CoverActiveDone();
		
	E_FixtureState.FIXTURE_EXTENSION_COVER_HOME:
		MS_CoverHome();
		
	E_FixtureState.FIXTURE_EXTENSION_COVER_HOME_DONE:
		MS_CoverHomeDone();
		
	E_FixtureState.FIXTURE_EXTENSION_CLAMP_HOLD:
		MS_ClampHold();
		
	E_FixtureState.FIXTURE_EXTENSION_CLAMP_HOLD_DONE:
		MS_ClampHoldDone();
		
	E_FixtureState.FIXTURE_EXTENSION_CLAMP_RELEASE:
		MS_ClampRelease();
		
	E_FixtureState.FIXTURE_EXTENSION_CLAMP_RELEASE_DONE:
		MS_ClampReleaseDone();
		
END_CASE
END_METHOD

END_FUNCTION_BLOCK

// ---- POUs/Universal Blocks/Fixture/FB_FixtureJig.TcPOU
(*
Copyrights	: Precision Systems Engineering
Author		: ADBO
Date		: 07/2022
Description	: This function block implements basic feature of Automatic FCQ fixture based on FB_UniversalFixture from PSE Shell library.
*)
FUNCTION_BLOCK FB_FixtureJig EXTENDS FB_UniversalFixture
VAR CONSTANT
	(* Fixture cover cylinder default setup *)
	sCOVER_NAME						: STRING := ':Jig';
	tCOVER_OPEN_TIMEOUT				: TIME	 := T#5S;
	tCOVER_CLOSE_TIMEOUT			: TIME	 := T#5S;
	tCOVER_MOVE_DELAY 				: TIME	 := T#0MS; //200MS
	sCOVER_HOME_SENSOR_MODULE		: STRING := 'Mainfold IO1';
	sCOVER_HOME_SENSOR_PORT_ID		: STRING := '1';
	sCOVER_ACTIVE_SENSOR_MODULE		: STRING := 'Mainfold IO1';
	sCOVER_ACTIVE_SENSOR_PORT_ID	: STRING := '2';
END_VAR
VAR
	eJigStateInit			: E_FixtureJigStateInit;	(*  *)
	eJigStateAbort			: E_FixtureJigStateAbort;	(*  *)
	eJigStateReset			: E_FixtureJigStateReset;	(*  *)
	
	(* Function blocks *)
	fbJig					: FB_DoubleCoilCylinder;	(*  *)
	
END_VAR

IF bFirstCycle THEN
	fbJig.MR_FirstCycle( 	sName 					:= CONCAT(STR1 := THIS^.sName, STR2 := sCOVER_NAME),
							sHomeSensorModuleType	:= sCOVER_HOME_SENSOR_MODULE,
							sHomeSensorPortID		:= sCOVER_HOME_SENSOR_PORT_ID,
							sActiveSensorModuleType	:= sCOVER_ACTIVE_SENSOR_MODULE,
							sActiveSensorPortID		:= sCOVER_ACTIVE_SENSOR_PORT_ID,
							tGoHomeTimeout 			:= tCOVER_CLOSE_TIMEOUT ,
							tGoActiveTimeout		:= tCOVER_OPEN_TIMEOUT,
							tDelay 					:= tCOVER_MOVE_DELAY);				
END_IF

(* Run parent main implementation *)
SUPER^();

(* Update status flags*)
bError := bError OR fbJig.Error;

(* Run product cover cylinder instance *)
fbJig();

PROPERTY JigSimulation : BOOL
GET
JigSimulation := fbJig.Simulation;
END_GET
SET
fbJig.Simulation := JigSimulation;
END_SET
END_PROPERTY

METHOD PROTECTED MS_Aborting
VAR_INPUT
END_VAR
CASE eJigStateAbort OF	
	(* Abort fixture product cover pusher *)
	FIXTURE_JIG_ABORT_JIG_PUSHER:
		fbJig.MR_Abort();
		IF NOT fbJig.Active THEN
			eFixtureStateAbort := UNIVERSAL_FIXTURE_ABORT_FILE_LOGGER;
			eJigStateAbort := FIXTURE_JIG_ABORT_DONE;
		END_IF
	
	(* Aborting done - run parent initialization *)
	FIXTURE_JIG_ABORT_DONE:
		SUPER^.MS_Aborting();
		
END_CASE
END_METHOD

METHOD PROTECTED MS_Close
VAR_INPUT
END_VAR
fbJig.MR_GoHome();
IF fbJig.PositionHome AND NOT fbJig.Busy THEN
	eFixtureState := UNIVERSAL_FIXTURE_METHOD_DONE;
END_IF
END_METHOD

METHOD PROTECTED MS_Initializing
VAR_INPUT
END_VAR
CASE eJigStateInit OF
	(* Initialize fixture product cover pusher *)
	FIXTURE_JIG_INIT_JIG_PUSHER:
		fbJig.MR_Init();
		
		IF fbJig.Active THEN
			IF eConnnectionType = UNIVERSAL_FIXTURE_CLIENT_CONNECTION THEN
				eFixtureStateInit := UNIVERSAL_FIXTURE_INIT_TCP_CLIENT;
			ELSIF eConnnectionType = UNIVERSAL_FIXTURE_SERVER_CONNECTION THEN
				eFixtureStateInit := UNIVERSAL_FIXTURE_INIT_TCP_SERVER;
			END_IF
			eJigStateInit := FIXTURE_JIG_INIT_DONE;
			
		END_IF
	
	(* Initializing done - run parent initialization*)
	FIXTURE_JIG_INIT_DONE:
		SUPER^.MS_Initializing();
		
END_CASE
END_METHOD

METHOD PROTECTED MS_Open
VAR_INPUT
END_VAR
fbJig.MR_GoActive();
IF fbJig.PositionActive AND NOT fbJig.Busy THEN
	eFixtureState := UNIVERSAL_FIXTURE_METHOD_DONE;
END_IF
END_METHOD

METHOD PROTECTED MS_Ready
VAR_INPUT
END_VAR
eFixtureState := UNIVERSAL_FIXTURE_IDLE;
END_METHOD

METHOD PROTECTED  MS_ReadyInitialized
VAR_INPUT
END_VAR
bBusy := FALSE;
eFixtureState := UNIVERSAL_FIXTURE_IDLE;
END_METHOD

METHOD PROTECTED MS_Reset
VAR_INPUT
END_VAR
CASE eJigStateReset OF
	FIXTURE_JIG_RESET_JIG_PUSHER:
		fbJig.MR_Reset();
		IF NOT fbJig.Error THEN
			eFixtureStateReset := UNIVERSAL_FIXTURE_RESETING_FILE_LOGGER;
			eJigStateReset := FIXTURE_JIG_RESET_DONE;
		END_IF
		
	FIXTURE_JIG_RESET_DONE:
		SUPER^.MS_Reset();
		
END_CASE
END_METHOD

PROPERTY ref_Jig : REFERENCE TO FB_DoubleCoilCylinder
GET
ref_Jig REF= fbJig;
END_GET
END_PROPERTY

PROPERTY SocketOpen : REFERENCE TO BOOL
GET
SocketOpen REF= fbJig.PositionActive;
END_GET
END_PROPERTY

END_FUNCTION_BLOCK

// ---- POUs/Universal Blocks/Fixture/FB_FixtureClamp.TcPOU
(*
Copyrights	: Precision Systems Engineering
Author		: ADBO
Date		: 07/2022
Description	: This function block is modyfication of standard FB_DoubleCoilCylinder.
It allows to operate double coil cylinder with only one sensor - active postion.
*)
FUNCTION_BLOCK FB_FixtureClamp EXTENDS FB_DoubleCoilCylinder

SUPER^();

METHOD MR_GoHome : BOOL
VAR_INPUT
END_VAR
IF eCylinderState = CYLINDER_IDLE AND piActiveSensor.In THEN
	bBusy := TRUE;
	bGoHome := TRUE;
	MR_GoHome := FALSE;
	
	eCylinderState := CYLINDER_GO_HOME;
	eCylinderGoHomeState := CYLINDER_MOVE_START_TRACKING;
	
	fbMachineLogger.MR_AddLogs(CONCAT(sName,' : home position requested'));	
	
ELSIF eCylinderState = CYLINDER_GO_HOME_DONE THEN
	bGoHome := FALSE;
	MR_GoHome := TRUE;
	
	fbMachineLogger.MR_AddLogs(CONCAT(sName,' : home position done'));	
	
END_IF
END_METHOD

METHOD PROTECTED MS_GoHome
poActiveValve.Out := FALSE;
poHomeValve.Out := TRUE;

CASE eCylinderGoHomeState OF
	CYLINDER_MOVE_START_TRACKING:
		IF NOT piActiveSensor.In THEN
			IF TIME_TO_INT(tDelay) = 0 THEN
				eCylinderGoHomeState := CYLINDER_MOVE_DONE;
			ELSE
				eCylinderGoHomeState := CYLINDER_MOVE_DELAY;
			END_IF
		END_IF
		
	CYLINDER_MOVE_DELAY:
		tonGoActiveDelay( IN := TRUE, PT := tDelay);
		
		IF tonGoActiveDelay.Q THEN
			tonGoActiveDelay( IN := FALSE );
			eCylinderGoHomeState := CYLINDER_MOVE_DONE;
		END_IF
		
	CYLINDER_MOVE_DONE:
		eCylinderState := CYLINDER_GO_HOME_DONE;
		
END_CASE
END_METHOD

END_FUNCTION_BLOCK

// ---- POUs/Universal Blocks/Fixture/PRG_FB_FcqFixture_Development_Test.TcPOU
(*
Copyrights	: Precision Systems Engineering
Author		: ADBO
Date		: 07/2022
Description: This program is used only for software development test of fixture FB only.
*)
PROGRAM PRG_FB_FcqFixture_Development_Test
VAR
	(* Generic flags *)
	bFirstCycle : BOOL := TRUE;
	
	(* Auxilary control buttons *)
	bInit					: BOOL;												(* Start initialization of fixture *)
	bAbort					: BOOL;												(* Start aborting of fixture *)
	bOpen					: BOOL;												(* Open fixture cover *)
	bClose					: BOOL;												(* Close fixture cover *)
	bReset					: BOOL;												(* Reset fixture *)
	bMeasure 				: BOOL;												(* Start measurement process *)
	bCoverHome				: BOOL;												(* Move fixture platform to home postion *)
	bCoverActive			: BOOL;												(* Move fixture platform to active postion *)
	bClampHold				: BOOL;												(* Hold product inside socket *)
	bClampRelease			: BOOL;												(* Realease product inside socket *)
	bCoverActiveAndJigOpen	: BOOL;												(* Opens fixture cover and moves platform to active position *)
	bCoverHomeAndJigClose	: BOOL;												(* Closes fixture cover and moves platform to home position *)
	bLoadNorm				: BOOL;												(* Send's trigger to UTU station to load product norm file *)
	                                                                			
	(* Parameters *)                                                			
	iSampleID				: UINT;												(*  *)
	bJigSimulation			: BOOL := FALSE;									(*  *)
	bCoverSimulation		: BOOL := FALSE;									(*  *)
	bClampSimulation 		: BOOL := FALSE;									(*  *)
	                                                                			
	(* Status *)                                                    			
	bActive					: REFERENCE TO BOOL;								(*  *)
	bBusy					: REFERENCE TO BOOL;								(*  *)
	bSocketOpen				: REFERENCE TO BOOL;								(*  *)
	iCurrentSampleID		: REFERENCE TO UDINT;								(*  *)
	bError					: REFERENCE TO BOOL;								(*  *)
	bCoverPositionActive 	: REFERENCE TO BOOL;								(*  *)
	bCoverPositionHome		: REFERENCE TO BOOL;								(*  *)
	bClampPositionHold		: REFERENCE TO BOOL;								(*  *)
	bNormLoaded				: REFERENCE TO BOOL;								(*  *)
	eMeasurementResult		: REFERENCE TO E_UniversalFixtureSampleResult;		(*  *)
	eMeasurementResultExt	: REFERENCE TO E_FixtureMeasurementResultExt;		(*  *)
	eState					: REFERENCE TO E_UniversalFixtureState;				(*  *)
	eStateExt				: REFERENCE TO E_FixtureState;						(*  *)
	
	(* Enums *)
	eFixtureTestState		: E_FixtureStateTest;								(*  *)
	
	(* Function blocks *)
	fbFixture 				: FB_Fixture;										(*  *)

END_VAR

IF bFirstCycle THEN
	bFirstCycle := FALSE;
	
	(* Assign initial parameters of fixture instance *)	
	fbFixture.MR_FirstCycle( 	sFixtureName		:= CONCAT(STR1 := sFIXTURE_NAME, STR2:= USINT_TO_STRING(1)),
											sHost 				:= '192.168.0.10',//CONCAT(STR1 := sFIXTURE_HOST, STR2:= '200'),//CONCAT(STR1 := sFIXTURE_HOST, STR2:= USINT_TO_STRING(iLoop)),
											sAmsNetID 			:= sFIXTURE_AMS_NET_ID,
											iPort 				:= iFIXTURE_PORT,
											tTimeout 			:= tFIXTURE_TIMEOUT,
											bUseLogger 			:= bFIXTURE_USE_LOGGER,
											bClientConnection	:= TRUE,//bFIXTURE_USE_CLIENT,
											sFileDir 			:= CONCAT(STR1:=sFIXTURE_FILE_DIR, STR2:= '\'),
											sFileName 			:= sFIXTURE_LOGGER_NAME,
											bCreateFileAtStart	:= TRUE,
											bAddHeader			:= TRUE,
											bAddTimeStamp		:= TRUE);
										
	(* Auxilary status flags references for watch*)
	bActive 				REF= fbFixture.Active;
	bBusy					REF= fbFixture.Busy;
	bSocketOpen 			REF= fbFixture.SocketOpen;
	iCurrentSampleID 		REF= fbFixture.SampleID;
	bError 					REF= fbFixture.Error;				
	bCoverPositionActive	REF= fbFixture.CoverPositionActive;
	bCoverPositionHome		REF= fbFixture.CoverPositionHome;
	bClampPositionHold		REF= fbFixture.ClampHold;
	eState					REF= fbFixture.State;
	eStateExt				REF= fbFixture.StateExt;
	bNormLoaded				REF= fbFixture.NormLoaded;
	eMeasurementResult		REF= fbFixture.SampleResult;
	eMeasurementResultExt	REF= fbFixture.MeasurementResultExt;
			
END_IF

(* Enable simulation of fixture pneumatic cylinders *)
fbFixture.JigSimulation := bJigSimulation;
fbFixture.CoverSimulation := bCoverSimulation;
fbFixture.ClampSimulation := bClampSimulation;
	
(* Generic control commands *)
IF bReset THEN
	bReset := FALSE;
	eFixtureTestState := FIXTURE_TEST_RESET;
			
ELSIF bAbort THEN
	fbFixture.MR_Abort();
	bAbort := FALSE;
	//eFixtureTestState := FIXTURE_TEST_ABORT;
	
END_IF

//IF fbFixture.State = UNIVERSAL_FIXTURE_UNINITIALIZED THEN
//	eFixtureTestState := FIXTURE_TEST_WAIT_FOR_COMMAND;
//END_IF

(* Manual tests state machine *)
CASE eFixtureTestState OF
	FIXTURE_TEST_WAIT_FOR_COMMAND:
		IF bInit THEN
			bInit := FALSE;
			eFixtureTestState := FIXTURE_TEST_INIT;
			
		ELSIF bOpen THEN
			bOpen := FALSE;
			eFixtureTestState := FIXTURE_TEST_OPEN;
			
		ELSIF bClose THEN
			bClose := FALSE;
			eFixtureTestState := FIXTURE_TEST_CLOSE;
			
		ELSIF bMeasure THEN
			bMeasure := FALSE;
			eFixtureTestState := FIXTURE_TEST_MEASURE;
			
		ELSIF bCoverHome THEN
			bCoverHome := FALSE;
			eFixtureTestState := FIXTURE_TEST_PLATFORM_HOME;
			
		ELSIF bCoverActive THEN
			bCoverActive := FALSE;
			eFixtureTestState := FIXTURE_TEST_PLATFORM_ACTIVE;
		
		ELSIF bClampHold THEN
			bClampHold := FALSE;
			eFixtureTestState := FIXTURE_TEST_PRODUCT_HOLD;
			
		ELSIF bClampRelease THEN
			bClampRelease := FALSE;
			eFixtureTestState := FIXTURE_TEST_PRODUCT_RELEASE;
			
		ELSIF bCoverActiveAndJigOpen THEN
			bCoverActiveAndJigOpen := FALSE;
			eFixtureTestState := FIXTURE_TEST_PLATFORM_ACTIVE_AND_OPEN;
			
		ELSIF bCoverHomeAndJigClose THEN
			bCoverHomeAndJigClose := FALSE;
			eFixtureTestState := FIXTURE_TEST_PLATFORM_HOME_AND_CLOSE;
			
		ELSIF bLoadNorm THEN
			bLoadNorm := FALSE;
			eFixtureTestState := FIXTURE_TEST_LOAD_NORM;
			
		END_IF
		
	FIXTURE_TEST_INIT:
		fbFixture.MR_Init();
		
		IF fbFixture.Active AND fbFixture.ref_Jig.Active AND fbFixture.ref_Clamp.Active AND fbFixture.ref_Cover.Active THEN
			eFixtureTestState := FIXTURE_TEST_WAIT_FOR_COMMAND;
		END_IF
	
	FIXTURE_TEST_OPEN:
		fbFixture.MR_Open();
		
		IF fbFixture.SocketOpen AND NOT fbFixture.Busy THEN
			eFixtureTestState := FIXTURE_TEST_WAIT_FOR_COMMAND;
		END_IF
	
	FIXTURE_TEST_CLOSE:
		fbFixture.MR_Close();
		
		IF NOT fbFixture.SocketOpen AND NOT fbFixture.Busy THEN
			eFixtureTestState := FIXTURE_TEST_WAIT_FOR_COMMAND;
		END_IF
	
	FIXTURE_TEST_MEASURE:
		fbFixture.MR_Measure(iSampleID := 0);
		
		IF NOT fbFixture.Busy THEN
			eFixtureTestState := FIXTURE_TEST_WAIT_FOR_COMMAND;
		END_IF
	
	FIXTURE_TEST_RESET:
		fbFixture.MR_Reset();
		
		IF NOT fbFixture.Error THEN
			eFixtureTestState := FIXTURE_TEST_WAIT_FOR_COMMAND;
		END_IF
	
	FIXTURE_TEST_ABORT:
		fbFixture.MR_Abort();
		
		IF NOT fbFixture.Active THEN
			eFixtureTestState := FIXTURE_TEST_WAIT_FOR_COMMAND;
		END_IF
	
	FIXTURE_TEST_PLATFORM_HOME:
		fbFixture.MR_CoverHome();
		
		IF fbFixture.CoverPositionHome AND NOT fbFixture.Busy THEN
			eFixtureTestState := FIXTURE_TEST_WAIT_FOR_COMMAND;
		END_IF
	
	FIXTURE_TEST_PLATFORM_ACTIVE:
		fbFixture.MR_CoverActive();
		
		IF fbFixture.CoverPositionActive AND NOT fbFixture.Busy THEN
			eFixtureTestState := FIXTURE_TEST_WAIT_FOR_COMMAND;
		END_IF
		
	FIXTURE_TEST_PRODUCT_HOLD:
		fbFixture.MR_ClampHold();
		
		IF fbFixture.ClampHold AND NOT fbFixture.Busy THEN
			eFixtureTestState := FIXTURE_TEST_WAIT_FOR_COMMAND;
		END_IF
	
	FIXTURE_TEST_PRODUCT_RELEASE:
		fbFixture.MR_ClampRelease();	
	
		IF NOT fbFixture.ClampHold AND NOT fbFixture.Busy THEN
			eFixtureTestState := FIXTURE_TEST_WAIT_FOR_COMMAND;
		END_IF
		
	FIXTURE_TEST_PLATFORM_ACTIVE_AND_OPEN:
		fbFixture.MR_CoverActiveAndJigOpen();
		
		IF fbFixture.CoverPositionActive AND fbFixture.SocketOpen AND NOT fbFixture.Busy THEN
			eFixtureTestState := FIXTURE_TEST_WAIT_FOR_COMMAND;
		END_IF
	
	FIXTURE_TEST_PLATFORM_HOME_AND_CLOSE:
		fbFixture.MR_CoverHomeAndJigClose();
		
		IF fbFixture.CoverPositionHome AND NOT fbFixture.SocketOpen AND NOT fbFixture.Busy THEN
			eFixtureTestState := FIXTURE_TEST_WAIT_FOR_COMMAND;
		END_IF
		
	FIXTURE_TEST_LOAD_NORM:
		//fbFixture.MR_LoadNorm( sProductType := 'E50', iProductQuantity := 100);
		
		IF fbFixture.NormLoaded THEN
			eFixtureTestState := FIXTURE_TEST_WAIT_FOR_COMMAND;
		END_IF
		
END_CASE

fbFixture();

END_PROGRAM

// ---- POUs/Universal Blocks/Robots/PRG_FB_CR800.TcPOU
PROGRAM PRG_FB_CR800
VAR
	fbCr800 : FB_CR800EtherCAT;
	
	(* HMI *)
	bInit 			: BOOL ;
	bAbort 			: BOOL ;
	bGoHome			: BOOL ;
	bGoAuto			: BOOL ;
	bCycleStop 		: BOOL ;
	bCyclePause		: BOOL ;
	bCycleRestore	: BOOL ;
	bDoAction		: BOOL ;
	bResetFBErr 	: BOOL ;
	bResetCR800Err	: BOOL ;
	bResetProgram 	: BOOL ;
	bUpdateRecipies	: BOOL ;
	btest 			: bool ;
	
	sState			: STRING ;
	sErrorName		: STRING ;
	
	iNumber			: UINT := 51;
	bRestoreAuto	: BOOL;
	bDoActionEnum	: BOOL;
	eRobotActions	: E_RobotActions ;
END_VAR

IF bInit THEN
	IF fbCr800.MR_Init() THEN
		bInit := FALSE ;
	END_IF
END_IF

IF bAbort THEN
	IF fbCr800.MR_Abort() THEN
		bAbort := FALSE ;
	END_IF
END_IF

IF bGoHome THEN
	IF fbCr800.MR_GoHome() THEN
		bGoHome := FALSE ;
	END_IF
END_IF

IF bGoAuto THEN
	IF fbCr800.MR_GoAuto() THEN
		bGoAuto := FALSE ;
	END_IF
END_IF

IF bCycleStop THEN
	IF fbCr800.MR_CycleStop() THEN
		bCycleStop := FALSE ;
	END_IF
END_IF

IF bCyclePause THEN
	IF fbCr800.MR_CyclePause() THEN
		bCyclePause := FALSE ;
	END_IF
END_IF

IF bCycleRestore THEN
	IF fbCr800.MR_RestoreCycle() THEN
		bCycleRestore := FALSE ;
	END_IF
END_IF

IF bDoAction THEN
	IF fbCr800.MR_DoAction(iActionNumber :=iNumber) THEN
		bDoAction := FALSE ;
	END_IF
END_IF

IF bResetFBErr THEN
	IF fbCr800.MR_Reset()  THEN
		bResetFBErr := FALSE ;
	END_IF
END_IF

IF bResetCR800Err THEN
	IF fbCr800.MR_ResetCR800Err()  THEN
		bResetCR800Err := FALSE ;
	END_IF
END_IF

IF bRestoreAuto THEN
	IF fbCr800.MR_RestoreAuto() THEN 
		bRestoreAuto := FALSE ;
	END_IF
END_IF

IF bDoActionEnum THEN
	IF fbCr800.MR_DoAction(iActionNumber :=E_RobotActions.PICK_AND_PLACE) THEN
		bDoActionEnum := FALSE ;
	END_IF
END_IF

IF bUpdateRecipies THEN
	IF fbCr800.MR_UpdateRecipies() THEN
		bUpdateRecipies := FALSE ;
	END_IF
END_IF

sState := fbCr800.MainStateMachine ;
sErrorName := fbCr800.Errorname ;

fbCr800();

END_PROGRAM

// ---- POUs/Universal Blocks/Utilities/Beckhoff UPS/PRG_FB_UpsCx20xx_Test.TcPOU
PROGRAM PRG_FB_UpsCx20xx_Test
VAR
	iSample		: INT := 10;
	fbUpsCX2020	: FB_UpsCx2xxx;
END_VAR

VAR PERSISTENT
	iSamplePersistent : INT := 10;
END_VAR

fbUpsCX2020.MR_FirstCycle( sName := 'Beckhoff UPS CX2020',
							sNetID := '',
							iPlcPort := 852,
							tTimeout := DEFAULT_ADS_TIMEOUT);

fbUpsCX2020();

END_PROGRAM

// ---- POUs/Universal Blocks/Utilities/Beckhoff UPS/PRG_FB_UpsCx50xx_Test.TcPOU
PROGRAM PRG_FB_UpsCx50xx_Test
VAR
	iSample		: INT := 10;
	fbUpsCX5000	: FB_UpsCx50xx;
END_VAR
VAR PERSISTENT
	iSamplePersistent : INT := 10;
END_VAR

fbUpsCX5000.MR_FirstCycle(	sName := 'Beckhoff UPS CX50xx',
							sNetID := '',
							iPlcPort := 852,
							tTimeout := DEFAULT_ADS_TIMEOUT);

fbUpsCX5000();

END_PROGRAM

// ---- POUs/Universal Blocks/Utilities/CSV Data Exchanger/PRG_FB_CSVDataExchanger_Test.TcPOU
PROGRAM PRG_FB_CSVDataExchanger_Test
VAR
	fbCSVDataExchanger	 		: FB_CSVDataExchanger;
	bFirstCycle 				: BOOL 		:= TRUE;
	
	sFileDir 					: STRING 	:= 'C:\TwinCAT\Tests\CSV_Reader\';
	sFileName 					: STRING 	:= 'Demo_Excel_File_FQC_Inputs_Test_2';
	sAmsNetId  					: STRING 	:= '';
	bAddHeader					: BOOL		:= FALSE;
	bCreateFile					: BOOL 		:= FALSE;
	bChangeSeparatorToComma		: BOOL 		:= FALSE;
	iMaxRowsNumber				: UDINT;
	iMaxColumnsNumber			: UDINT;
	
	bInit						: BOOL;
	bAbort						: BOOL;
	bReset						: BOOL;
	bSelectAll					: BOOL;
	bSelectRow					: BOOL;
	bSelectPath					: BOOL;
	bParseString				: BOOL;
			
	arrDatabase					: ARRAY[0..iMAX_CSV_ROWS - 1, 0..iMAX_CSV_COLUMNS - 1] OF STRING(iMAX_CSV_FIELD_LENGTH); (* Target PLC database *)	
	
	arrParsedString				: ARRAY[0..iMAX_CSV_COLUMNS - 1] OF STRING(iMAX_CSV_FIELD_LENGTH);	(* Target PLC database *)

	iColumnToSearch				: UDINT := 3;
	sValueToSearch			 	: WSTRING := "2";
	sRowResult				 	: STRING;
	
	
	iStateMachine				: USINT;
END_VAR

IF bFirstCycle THEN
	fbCSVDataExchanger.MR_FirstCycle(sFileDir 	:= sFileDir,
									sFileName 	:= sFileName,
									sAmsNetId 	:= '',
									bChangeSeparatorToComma := bChangeSeparatorToComma);									
	bFirstCycle := FALSE;
	
END_IF

IF bReset THEN
	bReset := FALSE;
	iStateMachine := 50;
	
ELSIF bAbort THEN
	bAbort := FALSE;
	iStateMachine := 60;

END_IF	

CASE iStateMachine OF
	0: 
		IF bInit THEN
			fbCSVDataExchanger.MR_Init();
			
			IF NOT fbCSVDataExchanger.Busy THEN
				bInit := FALSE;
				iStateMachine := 10;
				
			END_IF
		END_IF
		
	10: 
		IF bSelectAll THEN
			bSelectAll := FALSE;
			iStateMachine := 20;
		
		ELSIF bSelectRow THEN
			bSelectRow := FALSE;
			iStateMachine := 30;	

		ELSIF bSelectPath THEN
			bSelectPath := FALSE;
			iStateMachine := 40;	

		END_IF		
		
	20: 
		fbCSVDataExchanger.MR_SelectAll(iArrDataBaseAdr := ADR(arrDatabase));
		
		IF NOT fbCSVDataExchanger.Busy THEN
			iStateMachine := 10;
			
		END_IF
	
	30: 
		fbCSVDataExchanger.MR_SelectRow(iColumnToSearch := iColumnToSearch,
										sValueToSearch := WSTRING_TO_STRING(sValueToSearch),
										iArrParsedStringAdr := ADR(arrParsedString),
										sRowResult => sRowResult);
		
		IF NOT fbCSVDataExchanger.Busy THEN
			iStateMachine := 10;
			
		END_IF
	
	40:
		fbCSVDataExchanger.MR_SelectPath(sFileDir := sFileDir,
										sFileName := sFileName);
		
		IF NOT fbCSVDataExchanger.Busy THEN
			iStateMachine := 10;
			
		END_IF	

	50: 
		fbCSVDataExchanger.MR_Reset();
		
		IF NOT fbCSVDataExchanger.Busy THEN
			IF fbCSVDataExchanger.Active THEN
				iStateMachine := 10;
				
			ELSE
				iStateMachine := 0;
			
			END_IF
		END_IF
		
	60:
		fbCSVDataExchanger.MR_Abort();
	
		IF NOT fbCSVDataExchanger.Busy THEN
			iStateMachine := 0;
			
		END_IF
		
END_CASE

fbCSVDataExchanger();

END_PROGRAM

// ---- POUs/Universal Blocks/Utilities/File Logger/PRG_FB_FileLogger_Test.TcPOU
PROGRAM PRG_FB_FileLogger_Test
VAR
	bFirstCycle : BOOL := TRUE;
	
	sDirectoryForSimulation : STRING := 'C:\TwinCAT\Tests\';
	sFileDir 					: STRING 	:= 'C:\TwinCAT\Tests\\';
	sFileName 					: STRING 	:= 'Infile';
	
	fbFileLogger : FB_FileLogger;
	
	i 					: USINT;
	
	bInit				: BOOL;
	bAbort				: BOOL;
	bReset				: BOOL;
	
	bAddSingleLog 		: BOOL;
	bAddMaximumLoggs	: BOOL;
	bAddLogCommand		: BOOL;
	bSelectPath			: BOOL;
END_VAR

IF bFirstCycle THEN
	bFirstCycle := FALSE;
	fbFileLogger.MR_FirstCycle( sName		:= 'File Logger',
								sFileDir 	:= sDirectoryForSimulation,
								sFileName 	:= 'LoggerTest',
								sAmsNetId 	:= '',
								bAddTimeStamp := FALSE,
								bAddHeader := FALSE);
END_IF

IF bInit THEN
	fbFileLogger.MR_Init();
							
	IF fbFileLogger.Active THEN
		bInit := FALSE;
	END_IF
	
ELSIF bReset THEN
	fbFileLogger.MR_Reset();
	IF fbFileLogger.Busy THEN
		bReset := FALSE;
	END_IF
	
ELSIF bAbort THEN
	fbFileLogger.MR_Abort();
	IF NOT fbFileLogger.Active THEN
		bAbort := FALSE;
	END_IF
	
ELSIF bAddSingleLog THEN
	bAddSingleLog := FALSE;
	fbFileLogger.MR_AddLogs('Test message - 1');
	fbFileLogger.MR_AddLogs('Test message - 2');
	
ELSIF bSelectPath  THEN
	fbFileLogger.MR_SelectPath(sFileDir := sFileDir,
								sFileName := sFileName);
	
	IF NOT fbFileLogger.Busy THEN
		bSelectPath := FALSE;
		
	END_IF	

// Going outside buffer array (255) causes Windows blue screen
ELSIF bAddMaximumLoggs THEN
	FOR i := 0 TO 254 BY 1 DO 
		fbFileLogger.MR_AddLogs(CONCAT('Test message ',USINT_TO_STRING(i)));
		IF i = 254 THEN
			bAddMaximumLoggs := FALSE;
		END_IF
	END_FOR

END_IF

fbMachineTime( bEnable := TRUE);
fbFileLogger();
fbMachineLogger();

END_PROGRAM

// ---- POUs/Universal Blocks/Utilities/Recipes Manager/PRG_FB_RecipesManager_Test.TcPOU
PROGRAM PRG_FB_RecipesManager_Test
VAR
	bFirstCycle : BOOL := TRUE;
	
	bInit				: BOOL;						(*  *)
	bAbort				: BOOL;						(*  *)
	bCreate				: BOOL;						(*  *)
	bLoad				: BOOL;						(*  *)
	bLoadAndWritte		: BOOL;						(*  *)
	bRead				: BOOL;						(*  *)
	bReadAndSave		: BOOL;						(*  *)
	bRemove				: BOOL;						(*  *)
	bSave				: BOOL;						(*  *)
	bWritte				: BOOL;						(*  *)
	bGetRecipeCount		: BOOL;						(*  *)
	bGetRecipeNames		: BOOL;						(*  *)
	bGetVariableNames	: BOOL;						(*  *)
	bGetVariableValues	: BOOL;						(*  *)
	bReload				: BOOL;						(*  *)
	bRestore			: BOOL;						(*  *)
	bBackup				: BOOL;						(*  *)
	
	sLocalStoragePath	: STRING(512) := 'C:\TwinCAT\Tests\Recipes\';	(*  *)
	sRecipesDefinition	: STRING := 'Recipes';						(*  *)
	sRecipeName			: STRING := 'R1';							(*  *)

	fbRecipesControler	: FB_RecipesControler;
	
	rVar1 : REAL;
	rVar2 : REAL;
END_VAR

IF bFirstCycle THEN
	bFirstCycle := FALSE;
	fbRecipesControler.MR_FirstCycle(	sLocalStoragePath 	:= sLocalStoragePath,
										sRecipesDefinition	:= sRecipesDefinition,
										sDefaultRecipeName	:= sRecipeName);
	
END_IF

IF bInit THEN
	fbRecipesControler.MR_Init();
	IF fbRecipesControler.Active THEN
		bInit := FALSE;
	END_IF
	
ELSIF bAbort THEN
	fbRecipesControler.MR_Abort();
	IF NOT fbRecipesControler.Active THEN
		bAbort := FALSE;
	END_IF
	
ELSIF bCreate THEN
	IF fbRecipesControler.MR_Create(sRecipesDefinition, sRecipeName) THEN
		bCreate := FALSE;
	END_IF
	
ELSIF bLoad THEN
	IF fbRecipesControler.MR_Load(sRecipesDefinition, sRecipeName) THEN
		bLoad := FALSE;
	END_IF
	
ELSIF bLoadAndWritte THEN
	IF fbRecipesControler.MR_LoadAndWritte(sRecipesDefinition, sRecipeName) THEN
		bLoadAndWritte := FALSE;
	END_IF
	
ELSIF bRead THEN
	IF fbRecipesControler.MR_Read(sRecipesDefinition, sRecipeName) THEN
		bRead := FALSE;
	END_IF
	
ELSIF bReadAndSave THEN
	IF fbRecipesControler.MR_ReadAndSave(sRecipesDefinition, sRecipeName) THEN
		bReadAndSave := FALSE;
	END_IF
	
ELSIF bRemove THEN
	IF fbRecipesControler.MR_Remove(sRecipesDefinition, sRecipeName) THEN
		bRemove := FALSE;
	END_IF
	
ELSIF bSave THEN
	IF fbRecipesControler.MR_Save(sRecipesDefinition, sRecipeName) THEN
		bSave := FALSE;
	END_IF
	
ELSIF bWritte THEN
	IF fbRecipesControler.MR_Writte(sRecipesDefinition, sRecipeName) THEN
		bWritte := FALSE;
	END_IF
	
ELSIF bReload THEN
	IF fbRecipesControler.MR_Reload(sRecipeName,sRecipesDefinition) THEN
		bReload := FALSE;
	END_IF
	
ELSIF bGetRecipeNames THEN
	IF fbRecipesControler.MR_GetRecipesNames(sRecipesDefinition) THEN
		bGetRecipeNames := FALSE;
	END_IF
	
ELSIF bGetVariableNames THEN
	IF fbRecipesControler.MR_GetVariablesNames(sRecipesDefinition,sRecipeName) THEN
		bGetVariableNames := FALSE;
	END_IF
	
ELSIF bGetVariableValues THEN
	IF fbRecipesControler.MR_GetVariableValues(sRecipesDefinition,sRecipeName) THEN
		bGetVariableValues := FALSE;
	END_IF
	
END_IF

fbRecipesControler();

END_PROGRAM

// ---- POUs/Universal Blocks/Utilities/StringMerge/PRG_FUN_MergeStringsX_Test.TcPOU
PROGRAM PRG_FUN_MergeStringsX_Test
VAR
	sTestFunMergeLongStrings10	: STRING(2000);
	sTestFunMergeStrings10		: STRING(255);
	sTestFunMergeStrings5		: STRING(255);
END_VAR

sTestFunMergeLongStrings10 := FUN_MergeLongStrings10('1','2','3','4','5','6','7','8','9','10');
sTestFunMergeStrings10 := FUN_MergeStrings10('1','2','3','4','5','6','7','8','9','10');
sTestFunMergeStrings5 := FUN_MergeStrings5('1','2','3','4','5');

END_PROGRAM

// ---- POUs/Universal Blocks/Utilities/TXT Data Exchanger/PRG_FB_TXTDataExchanger_Test.TcPOU
PROGRAM PRG_FB_TXTDataExchanger_Test
VAR
	fbTXTDataExchanger	 		: FB_TXTDataExchanger;
	bFirstCycle 				: BOOL 		:= TRUE;
	
	sName						: STRING 	:= 'Txt data exchanger';
	sFileDir 					: STRING 	:= 'C:\TwinCAT\Tests\Recipes\';
	sFileName 					: STRING 	:= 'Infile';
	sAmsNetId  					: STRING 	:= '';
	bAddHeader					: BOOL		:= FALSE;
	bAddTimeStamp				: BOOL		:= FALSE;
	bCreateFileAtStart			: BOOL		:= FALSE;  
	
	bInit						: BOOL;
	bAbort						: BOOL;
	bReset						: BOOL;
	bAddMESCommand				: BOOL;
	bSearchForFile				: BOOL;
	bSelectPath					: BOOL;	
	
	sMachineID					: STRING	:= '32678';
	sOperatorID					: STRING	:= '0000025441';
	sPO							: STRING	:= '64822848';
	sProductItem				: STRING	:= '2159-3217599';
	bLogOn						: BOOL		:= TRUE;
	
	sSearchFileName				: STRING	:= 'R3.Recipes';
	bFileFound					: BOOL;
	
	iStateMachine				: USINT;
END_VAR

IF bFirstCycle THEN
	fbTXTDataExchanger.MR_FirstCycle(sName 	:= sName,
									sFileDir 	:= sFileDir,
									sFileName 	:= sFileName,
									sAmsNetId 	:= '',
									bCreateFileAtStart := bCreateFileAtStart,
									bAddHeader := bAddHeader,
									bAddTimeStamp := bAddTimeStamp);									
	bFirstCycle := FALSE;
	
END_IF

IF bReset THEN
	bReset := FALSE;
	iStateMachine := 50;
	
ELSIF bAbort THEN
	bAbort := FALSE;
	iStateMachine := 60;

END_IF	

CASE iStateMachine OF
	0: 
		IF bInit THEN
			fbTXTDataExchanger.MR_Init();
			
			IF NOT fbTXTDataExchanger.Busy THEN
				bInit := FALSE;
				iStateMachine := 10;
				
			END_IF
		END_IF
		
	10: 
		IF bAddMESCommand THEN
			bAddMESCommand := FALSE;
			iStateMachine := 20;
		
		ELSIF bSearchForFile THEN
			bSearchForFile := FALSE;
			iStateMachine := 30;	

		ELSIF bSelectPath THEN
			bSelectPath := FALSE;
			iStateMachine := 40;	

		END_IF		
		
	20: 
		fbTXTDataExchanger.MR_AddMESCommand(sMachineID := sMachineID,
											sOperatorID := sOperatorID,
											sPO := sPO,
											sProductItem := sProductItem,
											bLogOn := bLogOn);
		
		IF NOT fbTXTDataExchanger.Busy THEN
			iStateMachine := 10;
			
		END_IF
	
	30: 
		fbTXTDataExchanger.MR_SearchForFile(sSearchFileName := sSearchFileName, // Search in set path also
											bFileFound => bFileFound);
		
		IF NOT fbTXTDataExchanger.Busy THEN
			iStateMachine := 10;
			
		END_IF
	
	40:
		fbTXTDataExchanger.MR_SelectPath(sFileDir := sFileDir,
										sFileName := sFileName);
		
		IF NOT fbTXTDataExchanger.Busy THEN
			iStateMachine := 10;
			
		END_IF	

	50: 
		fbTXTDataExchanger.MR_Reset();
		
		IF NOT fbTXTDataExchanger.Busy THEN
			IF fbTXTDataExchanger.Active THEN
				iStateMachine := 10;
				
			ELSE
				iStateMachine := 0;
			
			END_IF
		END_IF
		
	60:
		fbTXTDataExchanger.MR_Abort();
	
		IF NOT fbTXTDataExchanger.Busy THEN
			iStateMachine := 0;
			
		END_IF
		
END_CASE

fbTXTDataExchanger();

END_PROGRAM

// ---- POUs/Universal Blocks/Vision/PRG_FB_Camera_Test.TcPOU
PROGRAM PRG_FB_Camera_Test
VAR
	bFirstCycle 			: BOOL := TRUE;
	fbFileLogger			: FB_FileLogger; 
	fbCamera				: FB_CognexCamera; 
	
	iState 					: USINT;
	
	bInit 					: BOOL;
	bAbort 					: BOOL;
	bReset					: BOOL;
	bGetConnections			: BOOL;
	bGetExpr				: BOOL;
	bGetFileList			: BOOL;
	bGetFile				: BOOL;	
	bGetOnline				: BOOL;	
	bGetValueEasyBuilder	: BOOL;	
	bGetValueSpreadsheet 	: BOOL;	
	bLoadFile				: BOOL;	
	bPutLive				: BOOL;	
	bPutPortnum				: BOOL;		
	bPutTimeout				: BOOL;	
	bPutUpdate				: BOOL;
	bPutWatch				: BOOL;
	bResetSystem			: BOOL;		
	bSetOnline				: BOOL;		
	bStoreFile				: BOOL;	
	bSetJob					: BOOL;
	bGetJob					: BOOL;
	bGetPosition			: BOOL;
	bImageTrigger			: BOOL;
	bGetValues				: BOOL;
	
	bError					: BOOL;
	iErrorID				: UDINT;
	
	sHost					: T_IPv4Addr;
	iPort					: UINT;
	
	sCellIndexExpr			: STRING 	:= 'A';
	iColumnExpr 			: INT		:= 0;
	iRowExpr 				: INT		:= 0;
	sEasyBuilderValuePositionX	: STRING	:= 'Pattern_1.Fixture.X';
	sEasyBuilderValuePositionY	: STRING	:= 'Pattern_1.Fixture.Y';
	sEasyBuilderValueRotation	: STRING	:= 'Pattern_1.Fixture.Angle';
	sEasyBuilderValueQuantity	: STRING	:= 'Pattern_1.Number_Found';
	
	iColumnValueSpreadsheet	: INT		:= 0;
	iRowValueSpreadsheet	: INT		:= 0;
	sLoadFileName			: STRING	:= 'Test.job';
	bEnableLiveAcquisition	: INT		:= 1;
	iPortNumber				: INT		:= 200;
	iTimeout				: INT		:= 20;	
	iUpdateNumber			: INT		:= 4;
	iColumnPut 				: INT		:= 0;
	iRowPut 				: INT		:= 0;
	iOutputEnable			: INT		:= 1;
	iJobNumber				: INT		:= 2;
	bSetCameraOnline		: INT		:= 1;
	sStoreFileName			: STRING	:= 'Test.job';
	
	lrPositionX				: LREAL;
	lrPositionY				: LREAL;
	lrRotation				: LREAL;

	lrValue1				: LREAL;
	lrValue2				: LREAL;
	lrValue3				: LREAL;
	lrValue4				: LREAL;
		
	sDirectoryForSimulation : STRING := 'C:\TwinCAT\Tests\';
	MR_ImageTrigger: INT;
	
	fbRobot					: FB_CR800EtherCAT;
END_VAR

(* Setting initial parameters *)
IF bFirstCycle THEN
	bFirstCycle := FALSE;
	fbCamera.MR_FirstCycle( 	sCameraName 	:= 'PShEll Test Camera',
								sClientHost		:= '192.168.0.151',
								sClientAmsNetID := '',
								iClientPort 	:= 23,
								tTimeout 		:= T#15S);
							
	fbFileLogger.MR_FirstCycle( sName		:= 'File Logger',
								sFileDir 	:= sDirectoryForSimulation,
								sFileName 	:= 'LoggerVisionTest',
								sAmsNetId 	:= '',
								bAddTimeStamp := TRUE,
								bAddHeader := TRUE);	
								
	iState := 0;
END_IF

bError := fbCamera.Error;
iErrorID := fbCamera.ErrorID;


(* Closing the client connection *)
IF bAbort THEN
	bAbort := FALSE;
	iState := 20;
END_IF

IF bReset THEN
	bReset := FALSE;
	iState := 30;
END_IF

CASE iState OF
	(* File logger initialization *)
	0:
		IF bInit THEN
				bInit := FALSE;		
				iState := 10;

		END_IF
		
	(* Client connection initialization *)
	10:
		fbCamera.MR_Init();
		IF fbCamera.Active THEN
			iState := 40;
		END_IF
		
	(* Client connection deinitialization *)
	20:
		fbCamera.MR_Abort();
		IF NOT fbCamera.Active THEN
			fbFileLogger.MR_Abort();
			IF NOT fbFileLogger.Active THEN
				iState := 0;	
			END_IF;
		END_IF
	
		
	30:	
		fbCamera.MR_Reset();
		IF NOT fbCamera.Busy THEN
			iState := 40;	
		END_IF
		
	(* Waiting for commands *)
	40:
		IF bGetConnections THEN
			bGetConnections := FALSE;
			iState := 50;
		ELSIF bGetExpr THEN
			bGetExpr := FALSE;
			iState := 60;	
		ELSIF bGetFileList THEN
			bGetFileList := FALSE;
			iState := 70;	
		ELSIF bGetFile THEN
			bGetFile := FALSE;
			iState := 80;	
		ELSIF bGetOnline THEN
			bGetOnline := FALSE;
			iState := 90;	
		ELSIF bGetValueEasyBuilder THEN
			bGetValueEasyBuilder := FALSE;
			iState := 100;	
		ELSIF bGetValueSpreadsheet THEN
			bGetValueSpreadsheet := FALSE;
			iState := 110;	
		ELSIF bLoadFile THEN
			bLoadFile := FALSE;
			iState := 120;	
		ELSIF bPutLive THEN
			bPutLive := FALSE;
			iState := 130;	
		ELSIF bPutPortnum THEN
			bPutPortnum := FALSE;
			iState := 140;	
		ELSIF bPutTimeout THEN
			bPutTimeout := FALSE;
			iState := 150;	
		ELSIF bPutUpdate THEN
			bPutUpdate := FALSE;
			iState := 160;	
		ELSIF bPutWatch THEN
			bPutWatch := FALSE;
			iState := 170;	
		ELSIF bResetSystem THEN
			bResetSystem := FALSE;
			iState := 180;	
		ELSIF bSetOnline THEN
			bSetOnline := FALSE;
			iState := 190;	
		ELSIF bStoreFile THEN
			bStoreFile := FALSE;
			iState := 200;	
		ELSIF bSetJob THEN
			bSetJob := FALSE;
			iState := 210;	
		ELSIF bGetJob THEN
			bGetJob := FALSE;
			iState := 220;	
		ELSIF bGetPosition THEN
			iState := 240;	
		ELSIF bImageTrigger THEN
			bImageTrigger := FALSE;
			iState := 240;	
		ELSIF bGetValues THEN
			iState := 240;	
		END_IF
		
	50:
		fbCamera.MR_GetConnections();
		IF NOT fbCamera.Busy THEN
			iState := 40;	
		END_IF

	60:
		
		fbCamera.MR_GetExpr(sCellIndexExpr,iColumnExpr,iRowExpr);
		IF NOT fbCamera.Busy THEN
			iState := 40;	
		END_IF		
	
	70:
		fbCamera.MR_GetFileList();
		IF NOT fbCamera.Busy THEN
			iState := 40;	
		END_IF
		
	80:
		fbCamera.MR_GetFile();
		IF NOT fbCamera.Busy THEN
			iState := 40;	
		END_IF

	90:
		fbCamera.MR_GetOnline();
		IF NOT fbCamera.Busy THEN
			iState := 40;	
		END_IF
		
	100:
		fbCamera.MR_GetValueEasyBuilder(sEasyBuilderValuePositionX);
		IF NOT fbCamera.Busy THEN
			iState := 40;	
		END_IF

	110:
		fbCamera.MR_GetValueSpreadsheet(iColumnValueSpreadsheet,iRowValueSpreadsheet);
		IF NOT fbCamera.Busy THEN
			iState := 40;	
		END_IF


	120:
		fbCamera.MR_LoadFile(sLoadFileName);
		IF NOT fbCamera.Busy THEN
			iState := 40;	
		END_IF

	130:
		fbCamera.MR_PutLive(bEnableLiveAcquisition);
		IF NOT fbCamera.Busy THEN
			iState := 40;	
		END_IF

	140:
		fbCamera.MR_PutPortnum(iPortNumber);
		IF NOT fbCamera.Busy THEN
			iState := 40;	
		END_IF

	150:
		fbCamera.MR_PutTimeout(iTimeout);
		IF NOT fbCamera.Busy THEN
			iState := 40;	
		END_IF

	160:
		fbCamera.MR_PutUpdate(iUpdateNumber);
		IF NOT fbCamera.Busy THEN
			iState := 40;	
		END_IF

	170:
		fbCamera.MR_PutWatch(iColumnPut,iRowPut,iOutputEnable);
		IF NOT fbCamera.Busy THEN
			iState := 40;	
		END_IF

	180:
		fbCamera.MR_ResetSystem();
		IF NOT fbCamera.Busy THEN
			iState := 40;	
		END_IF

	190:
		fbCamera.MR_SetOnline(bSetCameraOnline);
		IF NOT fbCamera.Busy THEN
			iState := 40;	
		END_IF

	200:
		fbCamera.MR_StoreFile(sStoreFileName);
		IF NOT fbCamera.Busy THEN
			iState := 40;	
		END_IF

	210:
		fbCamera.MR_SetJob(iJobNumber);
		IF NOT fbCamera.Busy THEN
			iState := 40;	
		END_IF

	220:
		fbCamera.MR_GetJob();
		IF NOT fbCamera.Busy THEN
			iState := 40;	
		END_IF
		
	230:
		fbCamera.MR_GetPosition(sPositionXVariable := sEasyBuilderValuePositionX,
								sPositionYVariable := sEasyBuilderValuePositionY,
								sRotationVariable := sEasyBuilderValueRotation,								
								lrPositionX => lrPositionX,
								lrPositionY => lrPositionY,
								lrRotation => lrRotation);
		IF NOT fbCamera.Busy THEN
			iState := 40;	
		END_IF
		
	240:
		fbCamera.MR_ImageTrigger();
		IF NOT fbCamera.Busy THEN
			IF bGetPosition THEN
				bGetPosition := FALSE;
				iState := 230;
			ELSIF bGetValues THEN
				bGetValues := FALSE;
				iState := 250;
			ELSIF NOT bGetPosition AND NOT bGetValues THEN	
				iState := 40;	
			END_IF	
		END_IF
		
	250:
	fbCamera.MR_GetValues(sVariable1 := sEasyBuilderValuePositionX,
							sVariable2 := sEasyBuilderValuePositionY,
							sVariable3 := sEasyBuilderValueRotation,		
							sVariable4 := sEasyBuilderValueQuantity,								
							lrValue1 => lrValue1,
							lrValue2 => lrValue2,
							lrValue3 => lrValue3,
							lrValue4 => lrValue4);
	IF NOT fbCamera.Busy THEN
		iState := 40;	
	END_IF
END_CASE

fbFileLogger();
fbCamera();

END_PROGRAM

// ---- POUs/Universal Blocks/XTS/FB_XtsStation.TcPOU
FUNCTION_BLOCK FB_XtsStation EXTENDS FB_XtsUniversalStation
VAR_INPUT
END_VAR
VAR_OUTPUT
END_VAR
VAR
END_VAR

IF bFirstCycle THEN
	(*
	Add MR_FirstCycle for declared station objects with initial setup.
	bFirstCycle bit is reseted by parent.
	*)
	
END_IF

(* Parent code *)
SUPER^();

(*
Add child main code here - handle declared station objects.
State machine is executed by parent code.
*)

METHOD PROTECTED M_RunningPerformProcess : BOOL
VAR_INPUT
END_VAR
(*
Add here code with process state machine e.g. perform action with robot and fixture.
Remember to set "_RunningPerformProcess := TRUE;" when te process is finished successfull - it will move parent state machine forward.
*)
(* Process simulation *)
tonProces( IN := TRUE, PT := T#3S);
IF tonProces.Q THEN
	tonProces( IN := FALSE);
	M_RunningPerformProcess := TRUE;
END_IF
END_METHOD

END_FUNCTION_BLOCK

// ---- POUs/Universal Blocks/XTS/PRG_XtsControlUnit_Test.TcPOU
PROGRAM PRG_XtsControlUnit_Test
VAR CONSTANT
	iNUMBER_OF_MOVERS 		: USINT := 2;
	iNUMBER_OF_STATIONS 	: USINT := 4;
	lrSTATION_POSITION_1 	: LREAL := 1875.0;
	lrSTATION_POSITION_2 	: LREAL := 1375.0;
	lrSTATION_POSITION_3 	: LREAL := 625.0;
	lrSTATION_POSITION_4 	: LREAL := 125.0;
	lrHOME_POSITION			: LREAL := 2150.0;
	lrRAIL_LENGTH			: LREAL := 2500.0;
END_VAR
VAR
	bFirstCycle	: BOOL := TRUE;
	iLoop		: USINT;
	
	bInit 	: BOOL;
	bHome 	: BOOL;
	bStart	: BOOL;
	bStop	: BOOL;
	bReset	: BOOL;
	bAbort	: BOOL;
	
	arrMover 			: ARRAY [0..iNUMBER_OF_MOVERS - 1] OF FB_XtsMover;
	arrStation			: ARRAY [0..iNUMBER_OF_STATIONS - 1] OF FB_XtsStation;
	
	fbXtsControlUnit 	: FB_XtsControlUnit;
	
	lrOverride			: LREAL;
	lrVelocity			: LREAL;
	lrAcceleration		: LREAL;
	lrDeceleration		: LREAL;
	lrJerk				: LREAL;
	lrJogVelocity		: LREAL;
	lrJogAcceleration	: LREAL;
	lrJogDeceleration	: LREAL;
	lrJogJerk			: LREAL;
	lrStopDeceleration	: LREAL;
	lrStopJerk			: LREAL;
	
	iState: INT;
	
	bFlag : BOOL;
END_VAR

(*  *)
IF bFirstCycle THEN
	bFirstCycle := FALSE;
	
	FOR iLoop := 0 TO iNUMBER_OF_MOVERS - 1 DO
		arrMover[iLoop].MR_FirstCycle( 	sName 				:= CONCAT(STR1 := 'Mover_',STR2 := USINT_TO_STRING(iLoop)),
										sMeasurementUnits 	:= 'mm',
										bModulo				:= TRUE);
	END_FOR
	
	arrStation[0].MR_FirstCycle(	sName 				:= 'Station 1',
									iStationID 			:= 0,
									ifNextStation 		:= arrStation[1],
									lrProcesPosition	:= lrSTATION_POSITION_1,
									lrWaitPosition		:= lrSTATION_POSITION_1 - 100.0,
									bWaitAfterStation	:= FALSE);
									
	arrStation[1].MR_FirstCycle(	sName 				:= 'Station 2',
									iStationID 			:= 1,
									ifNextStation 		:= arrStation[2],
									lrProcesPosition	:= lrSTATION_POSITION_2,
									lrWaitPosition		:= lrSTATION_POSITION_2 - 100.0,
									bWaitAfterStation	:= FALSE);
									
	arrStation[2].MR_FirstCycle(	sName 				:= 'Station 3',
									iStationID 			:= 2,
									ifNextStation 		:= arrStation[3],
									lrProcesPosition	:= lrSTATION_POSITION_3,
									lrWaitPosition		:= lrSTATION_POSITION_3 - 100.0,
									bWaitAfterStation	:= FALSE);
									
	arrStation[3].MR_FirstCycle(	sName 				:= 'Station 4',
									iStationID 			:= 3,
									ifNextStation 		:= arrStation[0],
									lrProcesPosition	:= lrSTATION_POSITION_4,
									lrWaitPosition		:= lrSTATION_POSITION_4 - 100.0,
									bWaitAfterStation	:= FALSE);
									
	fbXtsControlUnit.MR_FirstCycle( sName := 'XTS_Control_Unit:', lrRailLength := lrRAIL_LENGTH);
	
	FOR iLoop := 0 TO iNUMBER_OF_MOVERS - 1 DO
		fbXtsControlUnit.MR_AppendMover( ifMover := arrMover[iLoop]);
	END_FOR
	
	FOR iLoop := 0 TO iNUMBER_OF_STATIONS - 1 DO
		fbXtsControlUnit.MR_AppendStation( ifStation := arrStation[iLoop]);
	END_FOR
	
	lrOverride 			:= 100.0;
	lrVelocity 			:= 2000.0;
	lrAcceleration		:= 4000.0;
	lrDeceleration		:= 4000.0;
	lrJerk				:= 40000.0;
	
	lrJogVelocity 		:= 50.0;
	lrJogAcceleration	:= 1000.0;
	lrJogDeceleration	:= 1000.0;
	lrJogJerk			:= 10000.0;
	
	lrStopDeceleration	:= 4000.0;
	lrStopJerk			:= 40000.0;
	
	FOR iLoop := 0 TO iNUMBER_OF_MOVERS - 1 DO
		arrMover[iLoop].Override 			:= lrOverride;
		arrMover[iLoop].Velocity 			:= lrVelocity;
		arrMover[iLoop].SortingVelocity		:= 250.0;
		arrMover[iLoop].WorkVelocity		:= 2000.0;
		arrMover[iLoop].Acceleration 		:= lrAcceleration;
		arrMover[iLoop].Deceleration 		:= lrDeceleration;
		arrMover[iLoop].Jerk 				:= lrJerk;
		arrMover[iLoop].StopDeceleration	:= lrStopDeceleration;
		arrMover[iLoop].StopJerk			:= lrStopJerk;
	END_FOR
	
END_IF

(*  *)
IF bReset THEN
	bReset := FALSE;
	iState := 50;
ELSIF bAbort THEN
	bAbort := FALSE;
	iState := 60;
END_IF

(*  *)
CASE iState OF
	0:
		IF bInit THEN
			bInit := FALSE;
			iState := 10;
			
		ELSIF bHome THEN
			bHome := FALSE;
			iState := 20;
			
		ELSIF bStart THEN
			bStart := FALSE;
			iState := 30;
		
		ELSIF bStop THEN
			bStop := FALSE;
			iState := 40;

		END_IF

	10:
		bFlag := TRUE;
		
		FOR iLoop := 0 TO 5 DO
			arrStation[iLoop].MR_Init();
			bFlag := bFlag AND arrStation[iLoop].Active;
		END_FOR
		
		IF bFlag THEN
			iState := 15;
		END_IF
		
	15:
		fbXtsControlUnit.MR_Init();
		
		IF fbXtsControlUnit.Active THEN
			iState := 0;
		END_IF
	
	20:
		fbXtsControlUnit.MR_Home( lrHomePosition := lrHOME_POSITION);
		
		IF fbXtsControlUnit.IsHomed THEN
			iState := 0;
		END_IF
		
	30:
		fbXtsControlUnit.MR_Start();
		
		IF fbXtsControlUnit.Running THEN
			iState := 0;
		END_IF
		
	40:
		fbXtsControlUnit.MR_Stop();
		
		IF NOT fbXtsControlUnit.Running THEN
			iState := 0;
		END_IF
		
	50:
		fbXtsControlUnit.MR_Reset();
		
		IF NOT fbXtsControlUnit.Error THEN
			iState := 0;
		END_IF
		
	60:
		fbXtsControlUnit.MR_Abort();
		
		IF NOT fbXtsControlUnit.Active THEN
			iState := 0;
		END_IF
		
END_CASE

fbXtsControlUnit();

FOR iLoop := 0 TO iNUMBER_OF_STATIONS - 1 DO
	arrStation[iLoop]();
END_FOR

FOR iLoop := 0 TO iNUMBER_OF_MOVERS - 1 DO
	arrMover[iLoop]();
END_FOR

METHOD PROTECTED MS_Aborting
VAR_INPUT
END_VAR
(* 
Add here code to abort all station objects's e.g robots, axes, cylinders. 
At the end add "SUPER^.MS_Aborting();" to finish aborting.
*)

SUPER^.MS_Aborting();
END_METHOD

METHOD PROTECTED MS_Initializing
VAR_INPUT
END_VAR
(* 
Add here code to initialize all station objects's e.g robots, axes, cylinders. 
At the end add "eStateMachine := XTS_UNIVERSAL_STATION_READY_INITIALZIED;" to finish initialization.
*)

eStateMachine := XTS_UNIVERSAL_STATION_READY_INITIALZIED;
END_METHOD

METHOD PROTECTED MS_ReadyInitialized
VAR_INPUT
END_VAR
(*
Add code here if some internal parameters are needed to set after initialization or leave it default.
At the end add "eStateMachine := XTS_UNIVERSAL_STATION_IDLE;" to finish and go to IDLE state.
*)

eStateMachine := XTS_UNIVERSAL_STATION_IDLE;
END_METHOD

METHOD PROTECTED MS_Reset
VAR_INPUT
END_VAR
(*
Add here code to reset all station element's e.g robots, axes, cylinders.
*)

eStateMachine := XTS_UNIVERSAL_STATION_RESET_DONE;
END_METHOD

METHOD PROTECTED MS_Stop
VAR_INPUT
END_VAR
(*
Add here code to stop all station element's e.g robots, axes, cylinders, vision.
*)

eStateMachine := XTS_UNIVERSAL_STATION_STOP_DONE;
END_METHOD

METHOD PROTECTED MS_Uninitialized
VAR_INPUT
END_VAR
(* 
Add here code
At the end add "SUPER^.MS_Uninitialized();" to reset parent internal variables.
*)

SUPER^.MS_Uninitialized();
END_METHOD

END_PROGRAM

// ---- GlobalTextList.TcGTLO
TEXTLIST GlobalTextList
  331 = '%d'
  617 = '%f'
  976 = '%s'
  937 = '(* Add fields for process parameters according to machine specs*)'
  396 = '(* Add process parameters here *)'
  487 = 'Active Alarms'
  960 = 'Active alarms'
  649 = 'Active critical'
  488 = 'Active errors'
  582 = 'Active warrnings'
  755 = 'Add new recipe with current Values'
  518 = 'Admin'
  431 = 'Alarms'
  50 = 'All'
  917 = 'Change pass.'
  902 = 'Clear Alarm'
  349 = 'Clear All Alarms'
  277 = 'Close'
  410 = 'Close HMI'
  852 = 'Confirm Alarm'
  351 = 'Confirm All Alarms'
  197 = 'Current value:'
  507 = 'Errors'
  368 = 'Event history'
  86 = 'Event ID'
  606 = 'Event JSON Attribute'
  619 = 'Event Text'
  297 = 'Event Type'
  232 = 'Events history'
  231 = 'Export'
  77 = 'Export to file'
  464 = 'Label'
  715 = 'Lights'
  332 = 'Log In'
  198 = 'Log Out'
  372 = 'Maintenance'
  947 = 'Mechine running'
  417 = 'None'
  104 = 'Operator'
  615 = 'Page Auto'
  750 = 'Page Init'
  478 = 'Page Manual'
  20 = 'Page Manual Cylinders'
  5 = 'Page Manual Inputs'
  216 = 'Page Manual Motors'
  1674 = 'Page Manual Other'
  226 = 'Page Manual Outputs'
  946 = 'Page Manual Safety'
  554 = 'Page Recipes'
  979 = 'Page Uninitialized'
  495 = 'PageAuto'
  847 = 'Process'
  108 = 'Raise Alarm'
  156 = 'Raise Alarm 2'
  910 = 'Recipe variable 10:'
  311 = 'Recipe variable 11:'
  455 = 'Recipe variable 12:'
  766 = 'Recipe variable 13:'
  596 = 'Recipe variable 14:'
  883 = 'Recipe variable 15:'
  978 = 'Recipe variable 16:'
  334 = 'Recipe variable 17:'
  918 = 'Recipe variable 18:'
  273 = 'Recipe variable 19:'
  271 = 'Recipe variable 1:'
  567 = 'Recipe variable 20:'
  540 = 'Recipe variable 21:'
  977 = 'Recipe variable 22:'
  572 = 'Recipe variable 23:'
  324 = 'Recipe variable 24:'
  256 = 'Recipe variable 2:'
  323 = 'Recipe variable 3:'
  683 = 'Recipe variable 4:'
  342 = 'Recipe variable 5:'
  545 = 'Recipe variable 6:'
  718 = 'Recipe variable 7:'
  305 = 'Recipe variable 8:'
  51 = 'Recipe variable 9:'
  538 = 'Recipe1:'
  575 = 'Recipes'
  112 = 'Selected recipe value:'
  858 = 'Selected recipe:'
  289 = 'Send Alarm'
  698 = 'Send Message'
  909 = 'Service'
  853 = 'Set JSON'
  536 = 'Severity'
  586 = 'Step mode on'
  848 = 'Time Cleared'
  730 = 'Time Confirmed'
  9 = 'Time Raised'
  10 = 'Total active alarms'
  951 = 'Warnings'
END_TEXTLIST

// ---- VISUs/Platform/Pages/PageAuto.TcVIS
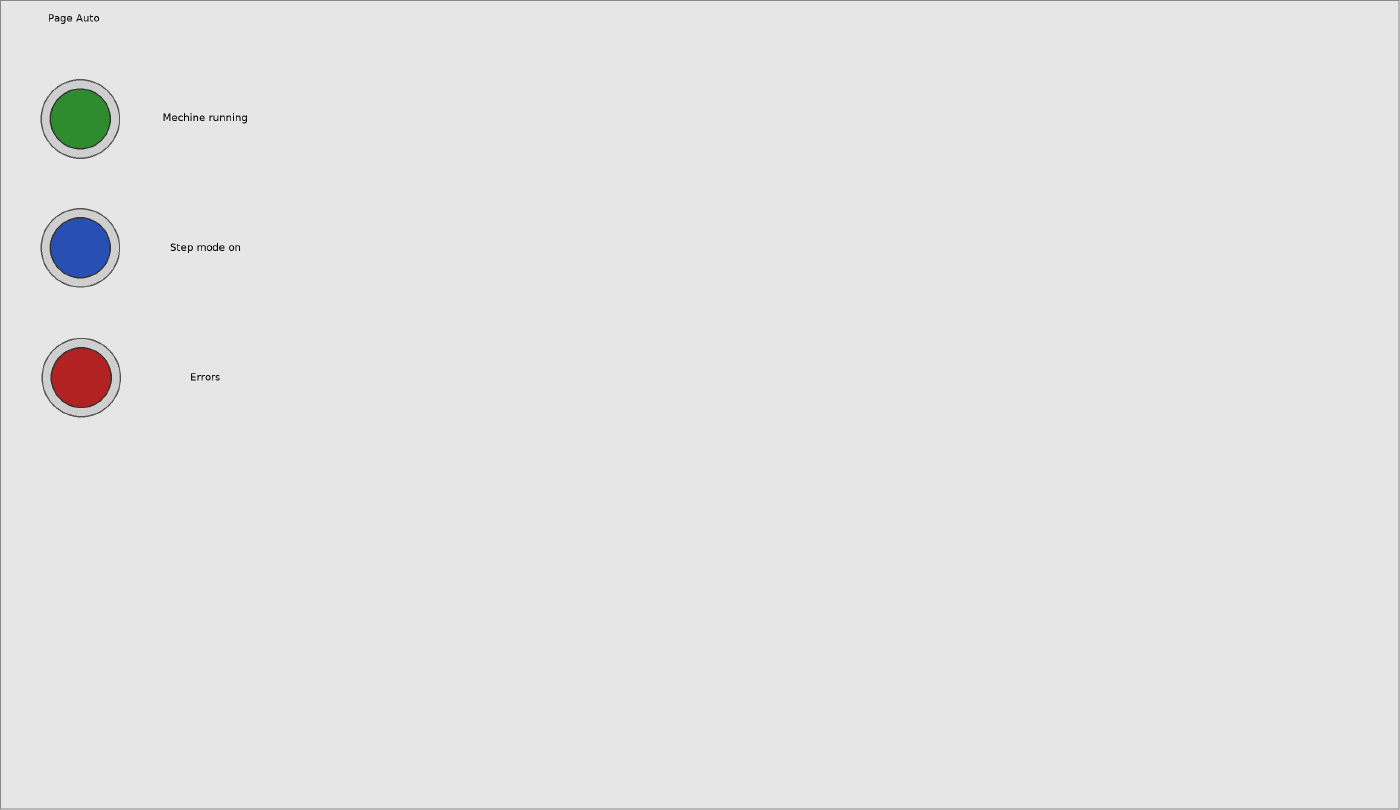
VISUALIZATION PageAuto  // 1520x880
    Label (5,5 150x30), "Page Auto"
    Label (148,113 150x30), "Mechine running"
    Label (148,254 150x30), "Step mode on"
    Lamp1 (37,79 100x100), variable: PRG_MachineControl.fbMachineControler.bRunning, style: Lamp-Lamp1-Green
    Lamp1 (37,219 100x100), variable: PRG_MachineControl.fbMachineControler.bStepMode, style: Lamp-Lamp1-Blue
    Lamp1 (38,360 100x100), variable: PRG_MachineControl.fbMachineControler.bError, style: Lamp-Lamp1-Red
    Label (148,395 150x30), "Errors"
END_VISUALIZATION

// ---- VISUs/Platform/Pages/PageInitializing.TcVIS
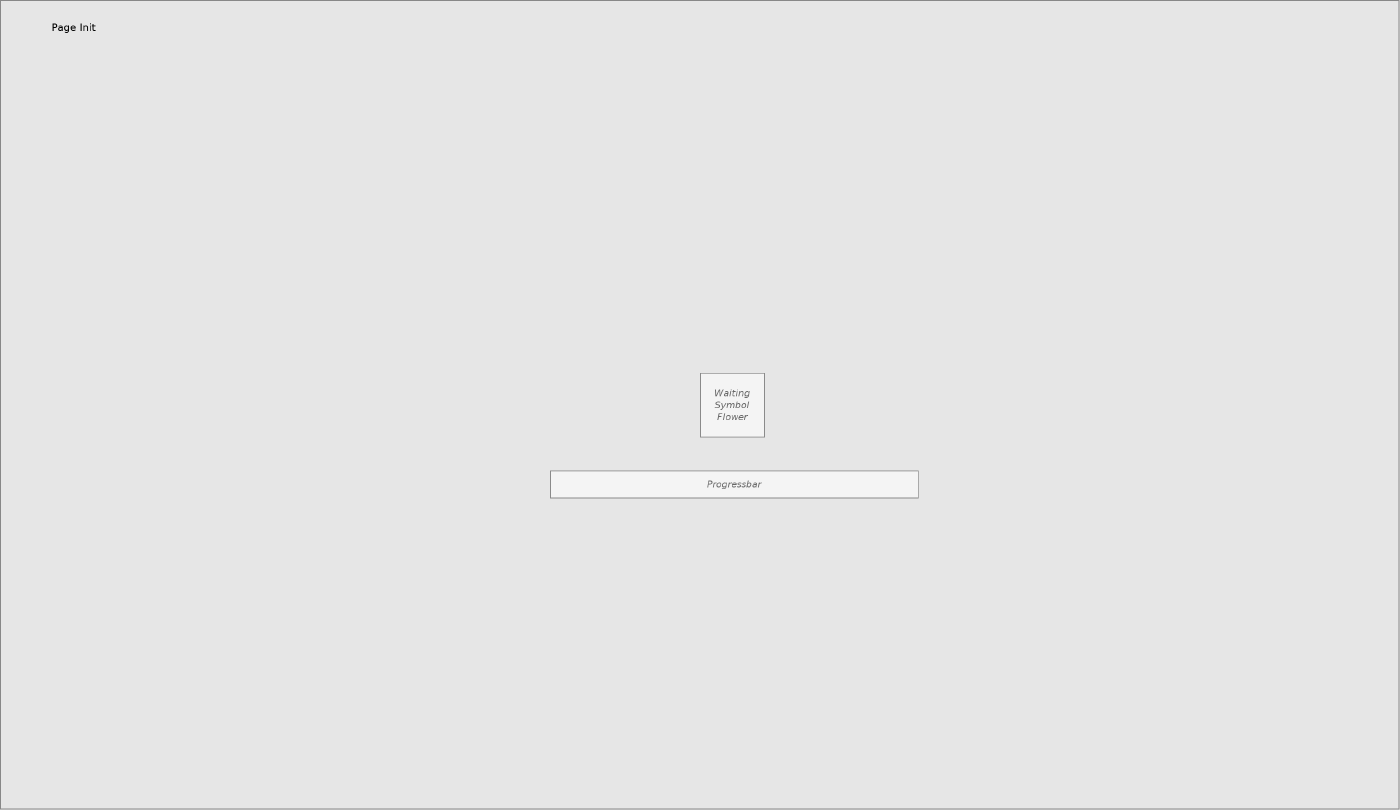
VISUALIZATION PageInitializing  // 1520x880
VAR_IN_OUT
	iProgressBar : USINT;
END_VAR
    Progressbar (597,511 400x30), variable: iProgressBar
    WaitingSymbolFlower (760,405 70x70)
    Label (5,15 150x30), "Page Init"
END_VISUALIZATION

// ---- VISUs/Platform/Pages/PageManualOther.TcVIS
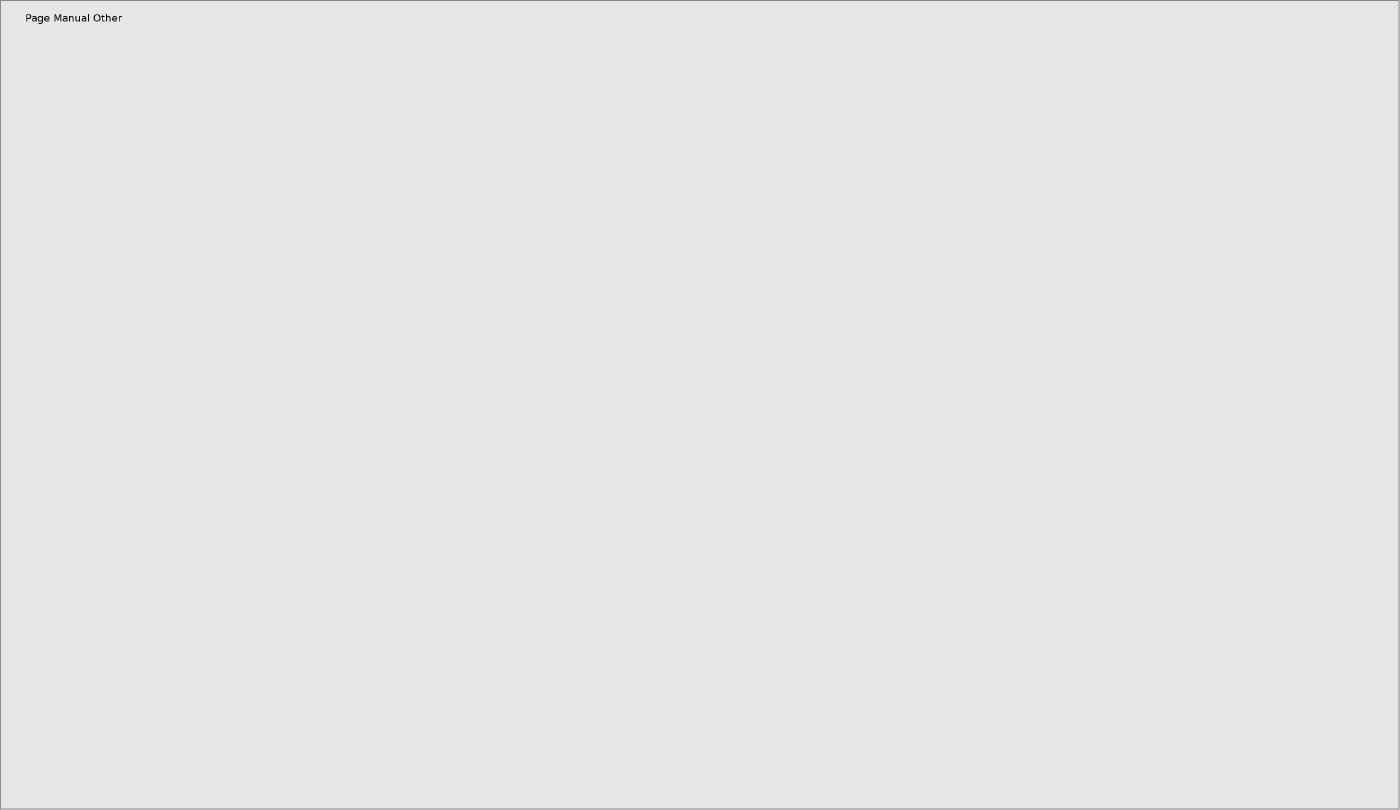
VISUALIZATION PageManualOther  // 1520x880
    Label (5,5 150x30), "Page Manual Other"
END_VISUALIZATION

// ---- VISUs/Platform/Pages/PageUninitialized.TcVIS
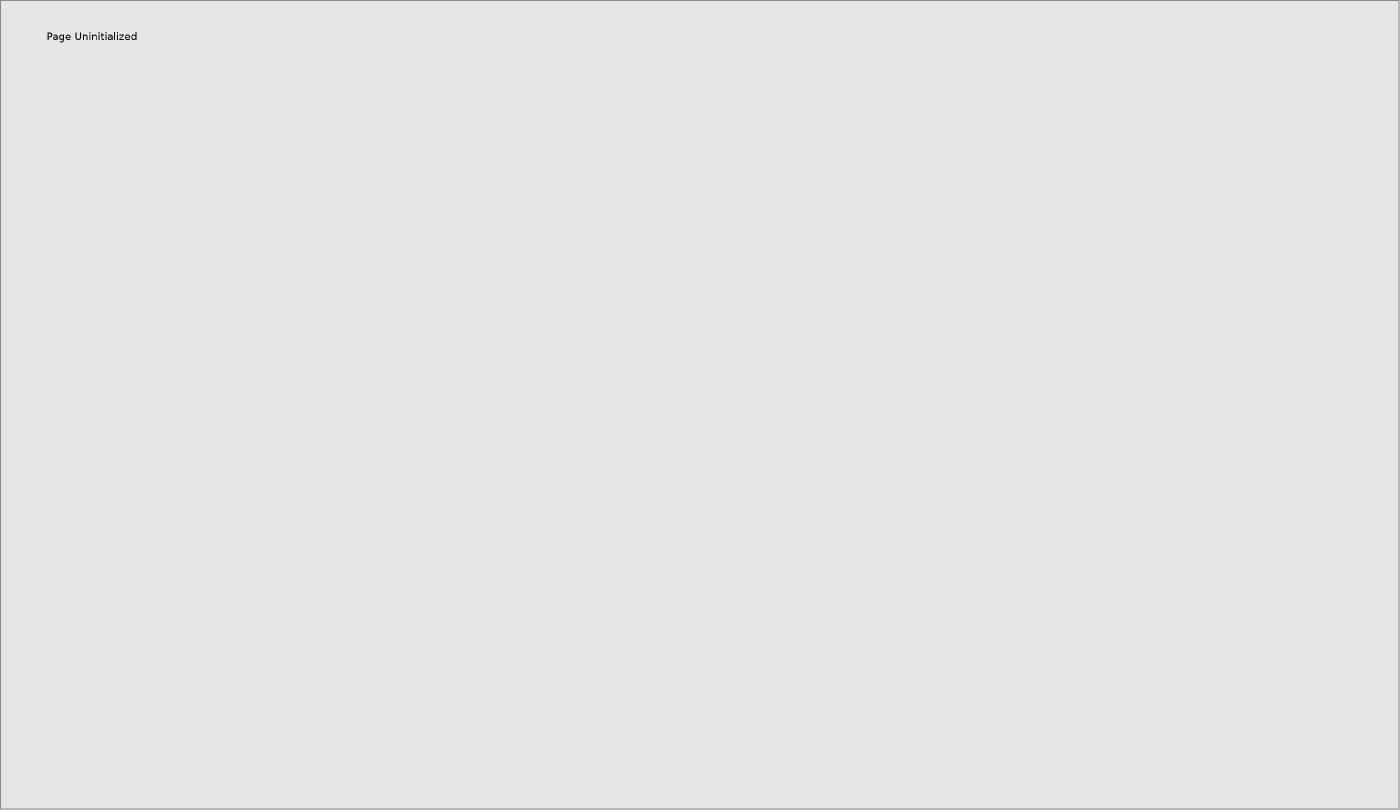
VISUALIZATION PageUninitialized  // 1520x880
    Label (25,25 150x30), "Page Uninitialized"
END_VISUALIZATION

